   "Q13.0" := "QCC除尘管道清洗阀";
   "Q13.1" := "QCC除尘清洗阀";
   "Q13.2" := "QSS输送管路清洗阀";
   "Q13.3" := "QLC料仓清洗阀";
   "Q13.4" := "QJR加热清洗阀";
   "Q13.5" := "QWK蜗壳清洗阀";//Q6.0
   "Q13.6" := "QCF出风高效清洗阀";
   "Q13.7" := "QZT主塔排水阀";

   "Q14.0" := "QSS输送管路排水阀";
   "Q14.1" := "QLC料仓清洗排水阀";
   "Q14.2" := "QSF送风机清洗阀";
   "Q14.3" := "QYF引风机清洗阀";
   "Q14.4" := "QYJ一级冷凝清洗阀";
   "Q14.5" := "QEJ二级冷凝清洗阀";
   "Q14.6" := "QSF送风机排水阀";
   "Q14.7" := "QYF引风机排水阀";

   "Q15.0" :="QYJ一级旋风振打锤" ;//主塔振打1
   "Q15.1" :="QYJ一级旋风振荡器" ;//主塔振打2
   "Q15.2" := "QEJ二级旋风振打锤";//主塔振打3
   "Q15.3" :="QZT主塔气锤4" ;//主塔振打4
   "Q15.4" :="QQZ前置水阀" ;//布袋振打1
   //"Q15.5" :="QSB设备振打" ;//布袋振打2
   (* "Q15.6" :="QBD布袋振打3" ;//布袋振打3
   "Q15.7" :="QBD布袋振打4" ;//布袋振打4 *)

   "Q15.6" :="QYH氧含仪隔断阀" ;//氧含仪隔断阀1
   "Q15.7" :="QHS回水隔断阀1" ;//这个空的



   //QW

   "QW100" := "QWFK放空比例调节阀";
   "QW102" := "QWJF进风加热比例调节阀";
   "QW104" := "QWHF回风加热比例调节阀";

   "QW108" := "QWSF送风机";
   "QW110" := "QWYF引风机";
   "QW112" := "QWLX离心雾化器";
   "QW114" := "QWJL进料泵";


   //IW 

   "IWJF进风流量计" := "IW100";
   "IWJL进料流量" := "IW102";
   "IWJF进风压差变送器" := "IW104";
   "IWCF出风高效压差变送器" := "IW106";

   "IWBD布袋压差变送器" := "IW108";
   "IWSS输送高效压差变送器" := "IW110";
   "IWJL进料压力" := "IW112";
   "IWTN塔内压力" := "IW114";

   "IWGD管道压力变送器" := "IW116";
   "IWJD进氮压力" := "IW118";
   "IWFK放空比例反馈" := "IW120";
   "IWJF进风加热比例反馈" := "IW122";

   "IWHF回风加热比例反馈" := "IW124";
   "IWWH雾化油压" := "IW126";
   "IWYH氧含仪1" := "IW128";
   "IWYH氧含仪2" := "IW130";

   //第二个模块
   "IWYJ一级溶剂液位计" := "IW132";
   "IWEJ二级溶剂液位计" := "IW134";
   "IWCW除雾溶剂液位计" := "IW136";
   "IWFD阀岛气压" := "IW138";

   "IWQZ前置水罐液位计" := "IW140";
   "IWBY备用2" := "IW142";
   "IWBY备用3" := "IW144";
   "IWBY备用4" := "IW146";


   //IW140-IW146空。
   "IWBY备用5" := "IW148";
   "IWSF送风机" := "IW150";
   "IWYF引风机" := "IW152";
   "IWLX离心雾化器" := "IW154";

   "IWJL进料泵" := "IW156";
   "IWBY备用6" := "IW158";
   "IWBY备用7" := "IW160";
   "IWBY备用8" := "IW162";
END_REGION
END_FUNCTION

FUNCTION_BLOCK "A8-通信心跳"   // FB31, SCL
{ S7_Optimized_Access := 'TRUE' }
VERSION : 0.1
// stored: AutoNumber true, IsIECCheckEnabled false, IsRetainMemResEnabled false, MemoryReserve 100, SetENOAutomatically false, UDAEnableTagReadback false
   VAR_INPUT
      XH信号超时报警 : Real := 120.0;   // SB设备写读与创造写对比,如果不同超时,即判断报警
   END_VAR
   VAR_OUTPUT
      设备未通信报警 : Bool;
   END_VAR
   VAR_IN_OUT
      SB设备写读 : Real;
      SB设备写 : Real;
      SB设备写检测 : Real;
   END_VAR
   VAR RETAIN
      MC脉冲切换时间 : Real := 20.0;   // 给写信号+1,创造不同，10秒切换一次
   END_VAR
   VAR
      XH信号不同超时报警 : Real := 120.0;   // SB设备写读与创造写对比,如果不同超时,即判断报警
      XH信号相同超时报警 : Real := 120.0;   // SB设备写读与创造写对比,如果相同超时,即判断报警
      TON1 { S7_SetPoint := 'True'} : TON_TIME;
      TON1ET { S7_SetPoint := 'True'} : Time;
      TON2 : TON_TIME;
      TON2ET { S7_SetPoint := 'True'} : Time;
      LS设备通延辅助1 { S7_SetPoint := 'True'} : Bool;
      LS设备通延辅助2 : Bool;
      LS通信脉冲读1 : Bool;
      LS通信脉冲读2 : Bool;
      LS设备读温比较 : Real;
      T1S : TON_TIME;
      YC1 { S7_SetPoint := 'True'} : Real;
   END_VAR
   VAR_TEMP
      "m" : Int;
   END_VAR
BEGIN
   IF "FirstScan" THEN
       RESET_TIMER(#TON1);
       RESET_TIMER(#TON2);
       #LS设备通延辅助1 := 0;
       #LS设备通延辅助2 := 0;
   END_IF;

   #XH信号不同超时报警:=#XH信号超时报警;
   #XH信号相同超时报警 := #XH信号超时报警;
   #MC脉冲切换时间 := 20;

   IF #T1S.Q AND #YC1<#MC脉冲切换时间 THEN
       #YC1 := #YC1 + 1;
   END_IF;

   IF #YC1 >= #MC脉冲切换时间 THEN
       #YC1 := 0;
   END_IF;

   IF #YC1 <= (#MC脉冲切换时间 - 10) THEN

       #LS通信脉冲读1 := 1;
       #LS通信脉冲读2 := 0;
   ELSE
       #LS通信脉冲读1 := 0;
       #LS通信脉冲读2 := 1;
   END_IF;

   IF #LS通信脉冲读1 THEN
       //冷水
       #LS设备读温比较 := #SB设备写读;
       #SB设备写检测 := #SB设备写 + 0.1;
       #TON1(IN := (ABS(#LS设备读温比较) <> ABS(#SB设备写检测)),
             PT := DINT_TO_TIME(REAL_TO_DINT(#XH信号不同超时报警 * 1000.0)),
             Q => #LS设备通延辅助1,
             ET => #TON1ET);

      #TON2(IN := (ABS(#LS设备读温比较) = ABS(#SB设备写检测)),
             PT := DINT_TO_TIME(REAL_TO_DINT(#XH信号相同超时报警 * 1000.0)),
             Q => #LS设备通延辅助2,
             ET => #TON2ET);

   END_IF;

   IF #LS通信脉冲读2 AND NOT #LS通信脉冲读1 THEN
       #SB设备写检测 := #SB设备写;
   END_IF;

   IF #LS设备通延辅助1 OR #LS设备通延辅助2  THEN
       #设备未通信报警 := 1;
   ELSE
       #设备未通信报警 := 0;
   END_IF;

   #T1S(IN := NOT #T1S.Q,
       PT := T#1S);
END_FUNCTION_BLOCK

FUNCTION_BLOCK "0-模拟量滤波"   // FB109, LAD
{ S7_Optimized_Access := 'TRUE' }
VERSION : 0.1
// stored: AutoNumber true, IsIECCheckEnabled false, IsRetainMemResEnabled false, MemoryReserve 100, SetENOAutomatically false, UDAEnableTagReadback false
   VAR_INPUT
      模拟量数据输入 : Int;
      "上限(工程量)" : Real;
      "下限(工程量)" : Real := 100.0;
      "采样时间间隔（秒）" : Real := 1.0;
      滤波强度 : Int := 10;
   END_VAR
   VAR_OUTPUT
      工程量数据输出 : Real;
      "工程量数据输出(滤波后)" : Real;
      Error_MAX : Bool;
      Error_MIN : Bool;
   END_VAR
   VAR
      AI : Int;
      "Time" : Time;
      T0 { S7_SetPoint := 'True'} : TON_TIME;
      T1 { S7_SetPoint := 'True'} : TON_TIME;
      P0 { S7_SetPoint := 'True'} : R_TRIG;
      LB { S7_SetPoint := 'True'} : Array[1..20] of Real;
      ZS : Real;
      N : Int;
      stat滤波强度 : Int;
   END_VAR
BEGIN

REGION Network 1 (SCL)
   #Time:=DINT_TO_TIME( REAL_TO_DINT( #"采样时间间隔（秒）"*1000.0)-10);
   #T0(IN:=NOT #T1.Q,
       PT:=#Time);
   #T1(IN:=#T0.Q,
       PT:=T#10MS);
   #P0(CLK:=#T0.Q);



   #AI := #模拟量数据输入;
   IF #AI<0 THEN
       #AI := 0;
       #Error_MIN := 1;
   ELSE
       #Error_MIN := 0;
       ;
   END_IF;

   IF #AI>27648 THEN
       #AI := 27648;
       #Error_MAX := 1;
   ELSE
       #Error_MAX := 0;
       ;
   END_IF;
   #stat滤波强度 := #滤波强度;
   IF #滤波强度 > 20 THEN
       #stat滤波强度 := 20;
   END_IF;
   IF #滤波强度 < 1 THEN
       #stat滤波强度 := 1;
   END_IF;

   IF #P0.Q THEN
       #工程量数据输出 := INT_TO_REAL(#AI) / 27648.0 * (#"上限(工程量)" - #"下限(工程量)") + #"下限(工程量)";
       FOR #N := #stat滤波强度 TO 2 BY -1 DO
           #LB[#N] := #LB[#N - 1];
           ;
       END_FOR;
       #LB[1] := #工程量数据输出;

       #ZS := 0;
       FOR #N := 1 TO #stat滤波强度 DO
           #ZS := #ZS + #LB[#N];
       END_FOR;


       #"工程量数据输出(滤波后)" := #ZS / #stat滤波强度;



   END_IF;
END_REGION
END_FUNCTION_BLOCK

FUNCTION_BLOCK "0-模拟量滤波简"   // FB86, SCL
{ S7_Optimized_Access := 'TRUE' }
VERSION : 0.1
// stored: AutoNumber true, IsIECCheckEnabled false, IsRetainMemResEnabled false, MemoryReserve 100, SetENOAutomatically false, UDAEnableTagReadback false
   VAR_INPUT
      输入 : Real;   // 转换后的模拟量输入端
      采集时间 : Time := T#200ms;   // 多长时间采集一次数据，单位ms
      模式 : Bool;   // false为算数平均滤波，true为切头尾平均滤波
   END_VAR
   VAR_OUTPUT
      输出 : Real;   // 滤波后的输出值
   END_VAR
   VAR_IN_OUT
      滤波强度 : Int := 3;   // 多少个数据平均一次
   END_VAR
   VAR
      T0 : TON_TIME;
      T1 { S7_SetPoint := 'True'} : TON_TIME;
      P { S7_SetPoint := 'True'} : R_TRIG;
      最小值 { S7_SetPoint := 'True'} : Real;
      最大值 : Real;
      中间寄存数值 : Array[0..30] of Real;
   END_VAR
   VAR_TEMP
      "a" : DInt;
      "b" : DInt;
      总和 : Real;
   END_VAR
BEGIN
   REGION 初始化
       #最大值 := #中间寄存数值[1];
       #最小值 := #中间寄存数值[1];
   END_REGION


   REGION 滤波强度限制
       IF #滤波强度 < 3 THEN
           #滤波强度 := 3;
       END_IF;
       IF #滤波强度 > 30 THEN
           #滤波强度 := 30;
       END_IF;
   END_REGION


   REGION 构速时钟脉冲
       #T0(IN := NOT #T1.Q,
           PT := #采集时间 - T#20MS);
       #T1(IN :=  #T0.Q,
           PT := T#20MS);
       #P(CLK := #T0.Q);
   END_REGION

   REGION 数据写入
       IF #P.Q THEN
           FOR #a := #滤波强度 TO 2 BY -1 DO //依次将输入数据存入到寄存数组中
               #中间寄存数值[#a] := #中间寄存数值[#a - 1];
           END_FOR;
           #中间寄存数值[1] := #输入;
       END_IF;
   END_REGION


   REGION 找最值以及计算总和
       FOR #b := 1 TO #滤波强度 DO
           IF #中间寄存数值[#b] > #最大值 THEN
               #最大值 := #中间寄存数值[#b];
           END_IF;
           IF #中间寄存数值[#b] < #最小值 THEN
               #最小值 := #中间寄存数值[#b];
           END_IF;
           #总和 := #总和 + #中间寄存数值[#b]; //计算总和
       END_FOR;
   END_REGION


   REGION 求平均以及输出
       IF #模式 = TRUE THEN
           #输出 := (#总和 - #最大值 - #最小值) / DINT_TO_REAL((#滤波强度) - 2);//切尾平均滤波后输出
       ELSE
           #输出 := #总和 / DINT_TO_REAL(#滤波强度);//算数平均输出
       END_IF;
   END_REGION
END_FUNCTION_BLOCK

FUNCTION_BLOCK "0-模拟量输入"   // FB35, SCL
{ S7_Optimized_Access := 'TRUE' }
VERSION : 0.1
// stored: AutoNumber true, IsIECCheckEnabled false, IsRetainMemResEnabled false, MemoryReserve 100, SetENOAutomatically false, UDAEnableTagReadback false
   VAR_INPUT
      模拟量数据输入 : Int;
      上限模拟 : Real := 27648.0;
      下限模拟 : Real := 5530.0;
      上限工程 : Real := 100.0;
      下限工程 : Real := 0.0;
      修正值 : Real;
      错误确认 : Bool;
      高高限工程量 : Real := 90.0;
      高限工程量 : Real := 80.0;
      低限工程量 : Real := 20.0;
      低低限工程量 : Real := 10.0;
      高高限位滤波时间设定 : Time := T#1s;
      高限位滤波时间设定 : Time := T#1s;
      低限位滤波时间设定 : Time := T#1s;
      低低限位滤波时间设定 : Time := T#1s;
      MODE : Byte := 16#1;   // 0报警输出不自动消除，1报警情况结束自动消除 2.高高或低低限位保持报警，其余自动确认报警
   END_VAR
   VAR_OUTPUT
      工程量数据输出 : Real;
      断线错误 : Bool;
      超过高高限位 : Bool;
      超过高限位 : Bool;
      低于低限位 : Bool;
      低于低低限位 : Bool;
   END_VAR
   VAR
      临时模拟量数据输入 : Real;
      缩放比例 : Real;
      T : Struct
         高高限位滤波时间 { S7_SetPoint := 'True'} : TON_TIME;
         高限位滤波时间 { S7_SetPoint := 'True'} : TON_TIME;
         低限位滤波时间 { S7_SetPoint := 'True'} : TON_TIME;
         低低限位滤波时间 { S7_SetPoint := 'True'} : TON_TIME;
      END_STRUCT;
   END_VAR
BEGIN
   #临时模拟量数据输入 := INT_TO_REAL(#模拟量数据输入);  //将模拟量输入转换为real类型
   // IF #临时模拟量数据输入 > #模拟量Max THEN
   //     #临时模拟量数据输入 := #模拟量Max;
   // END_IF;
   // IF #临时模拟量数据输入 < #模拟量Min THEN
   //     #临时模拟量数据输入 := #模拟量Min;
   // END_IF;
   #缩放比例 := (#上限工程 - #下限工程) / (#上限模拟 - #下限模拟);//算出实际值与模拟量的缩放比例
   #工程量数据输出 := (#模拟量数据输入 - #下限模拟) * #缩放比例 + #下限工程+#修正值;      //转换完成


   //2
   //
   IF (#临时模拟量数据输入 > 30000 OR #临时模拟量数据输入 < 4000 )
       AND NOT #错误确认 THEN
       #断线错误 := 1;
   ELSE
       #断线错误 := 0;
   END_IF;

   //3
   //

   #T.高高限位滤波时间(IN := #工程量数据输出 > #高高限工程量,
               PT := #高高限位滤波时间设定);
   IF #T.高高限位滤波时间.Q OR (#超过高高限位 AND (#MODE = 0 OR #MODE = 2)) AND NOT #错误确认 THEN

       #超过高高限位 := 1;
   ELSE
       #超过高高限位 := 0;
   END_IF;

   (* IF #超过高高限位 AND (#MODE = 0 OR #MODE = 2) AND NOT #错误确认 THEN
       #超过高高限位 := 1;
   ELSE
       #超过高高限位 := 0;
   END_IF; *)

   //4
   //
   #T.高限位滤波时间(IN := #工程量数据输出 >= #高限工程量,
              PT := #高限位滤波时间设定);
   IF #T.高限位滤波时间.Q OR (#超过高限位 AND #MODE = 0) AND NOT #错误确认 THEN
       #超过高限位 := 1;
   ELSE
       #超过高限位 := 0;
   END_IF;

   //5
   //
   #T.低限位滤波时间(IN := #工程量数据输出 <= #低限工程量,
              PT := #低限位滤波时间设定);

   IF #T.低限位滤波时间.Q OR (#低于低限位 AND #MODE = 0) AND NOT #错误确认 THEN
       #低于低限位 := 1;
   ELSE
       #低于低限位 := 0;
   END_IF;

   (* IF #低于低限位 AND #MODE=0 THEN
       #低于低限位 := 1;
   ELSE
       #低于低限位 := 0;
   END_IF; *)

   //6
   //
   #T.低低限位滤波时间(IN := #工程量数据输出 <= #低低限工程量,
               PT := #低低限位滤波时间设定);
   IF #T.低低限位滤波时间.Q OR (#低于低低限位 AND (#MODE = 0 OR #MODE = 2)) AND NOT #错误确认 THEN
       #低于低低限位 := 1;
   ELSE
       #低于低低限位 := 0;
   END_IF;

   (* IF #低于低低限位 AND (#MODE=0 OR #MODE=2) AND NOT #错误确认  THEN
       #低于低低限位 := 1;
   ELSE
       #低于低低限位 := 0;
   END_IF; *)
END_FUNCTION_BLOCK

FUNCTION_BLOCK "0-模拟量输入1PID"   // FB172, LAD
{ S7_Optimized_Access := 'TRUE' }
VERSION : 0.1
// stored: AutoNumber true, IsIECCheckEnabled false, IsRetainMemResEnabled false, MemoryReserve 100, SetENOAutomatically false, UDAEnableTagReadback false
   VAR_INPUT
      "仪表反馈值(模拟量)" : Int;
      积分P : Real := 0.5;
      微分I : Real := 0.5;
      "上限(模拟量)" : Real := 27648.0;
      "下限(模拟量)" : Real;
      "上限(工程量)" : Real := 200.0;
      "下限(工程量)" : Real;
      "设定补偿值(工程量)" : Real := 0.5;   // PID值快到达设定值时由于PID调节作用始终差一点才能到达设定值，所以用补偿的方式直接加上
      "设定目标值(工程量)" : Real := 100.0;
   END_VAR
   VAR_OUTPUT
      "仪表反馈值(工程量)" : Real;   // 由模拟量输入直接比例缩放转出的工程量，作用就是看一下显示
      "给定变频器(模拟量)" : Int;   // PID调节后的直接给变频器的模拟量值0-27648
      "PID调节输出值(工程量)" : Real;
   END_VAR
   VAR
      临时模拟量数据输入 : Real;
      缩放比例 : Real;
      实际模拟量 : Real;
      当前偏差 : Real;
      上一次偏差 : Real;
      输出控制量 : Real;
      PQW : Real;
   END_VAR
BEGIN

REGION Network 1 (SCL)
   //模拟量转换工程值
   #临时模拟量数据输入 := INT_TO_REAL(#"仪表反馈值(模拟量)");  //将模拟量输入转换为real类型
   #缩放比例 := (#"上限(工程量)" - #"下限(工程量)") / (#"上限(模拟量)" - #"下限(模拟量)");//算出实际值与模拟量的缩放比例
   #"仪表反馈值(工程量)" := (#"仪表反馈值(模拟量)"-#"下限(模拟量)") * #缩放比例+#"下限(工程量)";      //转换完成
   #当前偏差 := #"设定目标值(工程量)" - #"仪表反馈值(工程量)";

   //PID计算
   IF  #"设定补偿值(工程量)">ABS( #当前偏差) THEN
       #输出控制量 := 0;
   ELSIF #"设定补偿值(工程量)"<ABS( #当前偏差) THEN
       #输出控制量 := #积分P*(#当前偏差-#上一次偏差)+#微分I*#当前偏差;
   END_IF;

   #"PID调节输出值(工程量)":=#输出控制量;

   //上下限制
   IF #"PID调节输出值(工程量)"> #"上限(工程量)"THEN
       #"PID调节输出值(工程量)" := #"上限(工程量)";
   ELSIF #"PID调节输出值(工程量)"< #"下限(工程量)"THEN
       #"PID调节输出值(工程量)" := #"下限(工程量)";
   END_IF;


   //控制电机输出

   #上一次偏差 := #当前偏差;
   #PQW:=(#"PID调节输出值(工程量)"-#"下限(工程量)")/(#"上限(工程量)"-#"下限(工程量)")*#"上限(模拟量)";
   #"给定变频器(模拟量)" := REAL_TO_INT(#PQW);
END_REGION
END_FUNCTION_BLOCK

FUNCTION_BLOCK "0-模拟量输入2PID"   // FB79, SCL
{ S7_Optimized_Access := 'TRUE' }
VERSION : 0.1
// stored: AutoNumber true, IsIECCheckEnabled false, IsRetainMemResEnabled false, MemoryReserve 100, SetENOAutomatically false, UDAEnableTagReadback false
   VAR_INPUT
      AM : Bool := TRUE;   // 手动调节: 0,手动; 1,自动.
      ManualValue : Real;   // 手动调节输出值:0-100%.
      Enable : Bool;   // 自动调节使能. 1,启用; 0,不启用.
      Mode : Int := 1;   // 控制模式: 0,制热;1,制冷; 2,输出0.
      Setpoint : Real;   // 控制目标值
      Input : Real;   // 控制实际值
      ControlledObject_FB : Real;   // 受控对象实际值反馈(开度/频率...)
      Kp : Real;   // 比例系数(大于零实数)
      DeadZone : Real;   // 死区
      MAX : Real := 100.0;   // 上限
      MIN : Real;   // 下限
   END_VAR
   VAR_OUTPUT
      Output : Real;   // 受控对象输出值
   END_VAR
   VAR
      AutoValue : Real;
      output_Temp { ExternalAccessible := 'False'; ExternalVisible := 'False'; ExternalWritable := 'False'} : Real;
      RT_C : DInt;
   END_VAR
BEGIN
   IF  #AM AND #Enable THEN
       IF (#Mode=1) AND (ABS(#Input - #Setpoint) > #DeadZone) THEN
           #AutoValue := #ControlledObject_FB + #Kp * (#Input - #Setpoint) / 100;
       ELSIF (#Mode=0) AND (ABS(#Input - #Setpoint) > #DeadZone) THEN
           #AutoValue := #ControlledObject_FB - #Kp * (#Input - #Setpoint) / 100;
       ELSIF (#Mode=2) THEN
           #AutoValue := 0;
       ELSE
           #AutoValue := #ControlledObject_FB;
       END_IF;
   END_IF;

   IF NOT #AM THEN
       #output_Temp := #ManualValue;
   ELSE
       #output_Temp := #AutoValue;
   END_IF;

   IF #output_Temp >= #MAX THEN
       #Output := #MAX;
   ELSIF #output_Temp <= #MIN THEN
       #Output := #MIN;
   ELSE
       #Output := #output_Temp;
   END_IF;
END_FUNCTION_BLOCK

FUNCTION_BLOCK "0-模拟量输入压差"   // FB69, SCL
{ S7_Optimized_Access := 'TRUE' }
VERSION : 0.1
// stored: AutoNumber true, IsIECCheckEnabled false, IsRetainMemResEnabled false, MemoryReserve 100, SetENOAutomatically false, UDAEnableTagReadback false
   VAR_INPUT
      模拟量数据输入 : Int;
      上限模拟 : Real := 27648.0;
      下限模拟 : Real := 5530.0;
      上限工程 : Real := 100.0;
      下限工程 : Real := 0.0;
      修正值 : Real;
      错误确认 : Bool;
      高高限工程量 : Real := 90.0;
      高限工程量 : Real := 80.0;
      低限工程量 : Real := 20.0;
      低低限工程量 : Real := 10.0;
      高高限位滤波时间设定 : Time := T#1s;
      高限位滤波时间设定 : Time := T#1s;
      低限位滤波时间设定 : Time := T#1s;
      低低限位滤波时间设定 : Time := T#1s;
      MODE : Byte := 16#1;   // 0报警输出不自动消除，1报警情况结束自动消除 2.高高或低低限位保持报警，其余自动确认报警
   END_VAR
   VAR_OUTPUT
      工程量数据输出 : Real;
      断线错误 : Bool;
      超过高高限位 : Bool;
      超过高限位 : Bool;
      低于低限位 : Bool;
      低于低低限位 : Bool;
   END_VAR
   VAR_IN_OUT
      风机 : Bool;
   END_VAR
   VAR
      临时模拟量数据输入 : Real;
      缩放比例 : Real;
      T : Struct
         高高限位滤波时间 { S7_SetPoint := 'True'} : TON_TIME;
         高限位滤波时间 { S7_SetPoint := 'True'} : TON_TIME;
         低限位滤波时间 { S7_SetPoint := 'True'} : TON_TIME;
         低低限位滤波时间 { S7_SetPoint := 'True'} : TON_TIME;
      END_STRUCT;
   END_VAR
BEGIN
   #临时模拟量数据输入 := INT_TO_REAL(#模拟量数据输入);  //将模拟量输入转换为real类型
   // IF #临时模拟量数据输入 > #模拟量Max THEN
   //     #临时模拟量数据输入 := #模拟量Max;
   // END_IF;
   // IF #临时模拟量数据输入 < #模拟量Min THEN
   //     #临时模拟量数据输入 := #模拟量Min;
   // END_IF;
   #缩放比例 := (#上限工程 - #下限工程) / (#上限模拟 - #下限模拟);//算出实际值与模拟量的缩放比例
   #工程量数据输出 := (#模拟量数据输入 - #下限模拟) * #缩放比例 + #下限工程+#修正值;      //转换完成


   //2
   //
   IF (#临时模拟量数据输入 > 30000 OR #临时模拟量数据输入 < 4000 OR #断线错误)
       AND NOT #错误确认 THEN
       #断线错误 := 1;
   ELSE
       #断线错误 := 0;
   END_IF;

   //3
   //

   #T.高高限位滤波时间(IN := #工程量数据输出 > #高高限工程量,
               PT := #高高限位滤波时间设定);
   IF #T.高高限位滤波时间.Q OR (#超过高高限位 AND (#MODE = 0 OR #MODE = 2)) AND NOT #错误确认 THEN

       #超过高高限位 := 1;
   ELSE
       #超过高高限位 := 0;
   END_IF;

   (* IF #超过高高限位 AND (#MODE = 0 OR #MODE = 2) AND NOT #错误确认 THEN
       #超过高高限位 := 1;
   ELSE
       #超过高高限位 := 0;
   END_IF; *)

   //4
   //
   #T.高限位滤波时间(IN := #工程量数据输出 >= #高限工程量,
              PT := #高限位滤波时间设定);
   IF #T.高限位滤波时间.Q OR (#超过高限位 AND #MODE = 0) AND NOT #错误确认 THEN
       #超过高限位 := 1;
   ELSE
       #超过高限位 := 0;
   END_IF;

   //5
   //
   #T.低限位滤波时间(IN := #工程量数据输出 <= #低限工程量,
              PT := #低限位滤波时间设定);

   IF #T.低限位滤波时间.Q OR (#低于低限位 AND #MODE = 0) AND #风机 AND NOT #错误确认 THEN
       #低于低限位 := 1;
   ELSE
       #低于低限位 := 0;
   END_IF;

   (* IF #低于低限位 AND #MODE=0 THEN
       #低于低限位 := 1;
   ELSE
       #低于低限位 := 0;
   END_IF; *)

   //6
   //
   #T.低低限位滤波时间(IN := #工程量数据输出 <= #低低限工程量,
               PT := #低低限位滤波时间设定);
   IF #T.低低限位滤波时间.Q OR (#低于低低限位 AND (#MODE = 0 OR #MODE = 2)) AND NOT #错误确认 THEN
       #低于低低限位 := 1;
   ELSE
       #低于低低限位 := 0;
   END_IF;

   (* IF #低于低低限位 AND (#MODE=0 OR #MODE=2) AND NOT #错误确认  THEN
       #低于低低限位 := 1;
   ELSE
       #低于低低限位 := 0;
   END_IF; *)
END_FUNCTION_BLOCK

FUNCTION_BLOCK "1-模拟量输出1"   // FB75, SCL
{ S7_Optimized_Access := 'TRUE' }
VERSION : 0.1
// stored: AutoNumber true, IsIECCheckEnabled false, IsRetainMemResEnabled false, MemoryReserve 100, SetENOAutomatically false, UDAEnableTagReadback false
   VAR_INPUT
      HMI上限 : Real;
      HMI下限 : Real;
      PLC上限 : Int;
      PLC下限 : Int;
   END_VAR
   VAR_IN_OUT
      PLC调控 : Int;
      HMI设定 : Real;
   END_VAR
   VAR
      DBD1 : Real;
   END_VAR
BEGIN
   #DBD1 := NORM_X_REAL(MIN := #HMI下限, VALUE := #HMI设定, MAX := #HMI上限);
   #PLC调控 := SCALE_X_INT(MIN := #PLC下限, VALUE := #DBD1, MAX := #PLC上限);
END_FUNCTION_BLOCK

FUNCTION_BLOCK "1-模拟量输出2"   // FB77, SCL
{ S7_Optimized_Access := 'TRUE' }
VERSION : 0.1
// stored: AutoNumber true, IsIECCheckEnabled false, IsRetainMemResEnabled false, MemoryReserve 100, SetENOAutomatically false, UDAEnableTagReadback false
   VAR_INPUT
      R_Max : Real;
      R_Min : Real;
      R_Value : Real;
   END_VAR
   VAR_OUTPUT
      I_ChValue : Int;
   END_VAR
BEGIN
   (**)
   #I_ChValue := REAL_TO_INT((#R_Value - #R_Min) / (#R_Max - #R_Min) * 27648.0);
END_FUNCTION_BLOCK

FUNCTION_BLOCK "3-延时开关M"   // FB78, SCL
{ S7_Optimized_Access := 'TRUE' }
VERSION : 0.1
// stored: AutoNumber true, IsIECCheckEnabled false, IsRetainMemResEnabled false, MemoryReserve 100, SetENOAutomatically false, UDAEnableTagReadback false
   VAR_INPUT
      B_IN : Bool;   // 启动/关闭信号输入
      T_IN : Int;   // 延时时间(单位:分)
      B_Status : Bool;   // 运行状态
   END_VAR
   VAR_OUTPUT
      B_OUT : Bool;   // 启动/关闭信号输出
   END_VAR
   VAR
      RT1 { S7_SetPoint := 'True'} : R_TRIG;   // 计时_1S
      i : UDInt;
   END_VAR
BEGIN
   (*水泵关机延时功能:
       1.立即开机
       2.延时I_IN分钟后关闭
       3.延时关机期间如果水泵手动/其他原因关闭,延时时间清零,立即关闭
   *)

   #RT1(CLK:="Clock_1Hz");

   IF NOT #B_IN THEN
       IF #RT1.Q THEN
           #i += 1;
       END_IF;
   ELSE
       #i := 0;
   END_IF;

   IF #B_IN THEN
       #B_OUT := 1;    //立即开
   ELSIF NOT #B_IN AND #i >= #T_IN * 60 THEN    //延时关
       #B_OUT := 0;
   ELSIF NOT #B_IN AND #i < #T_IN * 60 AND  #B_Status THEN  //延时关机期间如果水泵手动/其他原因关闭,延时时间清零,立即关闭
       #B_OUT := 0;
   END_IF;
END_FUNCTION_BLOCK

FUNCTION_BLOCK "3-延时开关S"   // FB73, SCL
{ S7_Optimized_Access := 'TRUE' }
VERSION : 0.1
// stored: AutoNumber true, IsIECCheckEnabled false, IsRetainMemResEnabled false, MemoryReserve 100, SetENOAutomatically false, UDAEnableTagReadback false
   VAR_INPUT
      B_IN : Bool;   // 启动/关闭信号输入
      T_IN : Int;   // 延时时间(单位:秒)
      B_Status : Bool;   // 运行状态
   END_VAR
   VAR_OUTPUT
      B_OUT : Bool;   // 启动/关闭信号输出
   END_VAR
   VAR
      R_TRIG_1 { S7_SetPoint := 'True'} : R_TRIG;   // 计时_1S
      i : UDInt;
   END_VAR
BEGIN
   (*水泵关机延时功能:
       1.立即开机
       2.延时I_IN分钟后关闭
       3.延时关机期间如果水泵手动/其他原因关闭,延时时间清零,立即关闭
   *)

   #R_TRIG_1(CLK:="Clock_1Hz");

   IF NOT #B_IN THEN
       IF #R_TRIG_1.Q THEN
           #i += 1;
       END_IF;
   ELSE
       #i := 0;
   END_IF;

   IF #B_IN THEN
       #B_OUT := 1;    //立即开
   ELSIF NOT #B_IN AND #i >= #T_IN  THEN    //延时关
       #B_OUT := 0;
   ELSIF NOT #B_IN AND #i < #T_IN  AND  #B_Status THEN  //延时关机期间如果水泵手动/其他原因关闭,延时时间清零,立即关闭
       #B_OUT := 0;
   END_IF;
END_FUNCTION_BLOCK

FUNCTION_BLOCK "4-点斜率输入->输出"   // FB64, LAD
{ S7_Optimized_Access := 'TRUE' }
VERSION : 0.1
// stored: AutoNumber true, IsIECCheckEnabled false, IsRetainMemResEnabled false, MemoryReserve 100, SetENOAutomatically false, UDAEnableTagReadback false
   VAR_INPUT
      sr输入ok : Real;
   END_VAR
   VAR_OUTPUT
      sc输出ok : Int;
   END_VAR
   VAR_IN_OUT
      sr输入1 : Real;
      sc输出1 : Real;
      sr输入2 : Real;
      sc输出2 : Real;
   END_VAR
BEGIN

REGION Network 1 (SCL)


   #sc输出ok := REAL_TO_INT(((#sc输出2 - #sc输出1) / (#sr输入2 - #sr输入1)) * #sr输入ok);
END_REGION
END_FUNCTION_BLOCK

FUNCTION_BLOCK "4-点斜率输出->输入"   // FB68, LAD
{ S7_Optimized_Access := 'TRUE' }
VERSION : 0.1
// stored: AutoNumber true, IsIECCheckEnabled false, IsRetainMemResEnabled false, MemoryReserve 100, SetENOAutomatically false, UDAEnableTagReadback false
   VAR_INPUT
      sc输出ok : Int;
   END_VAR
   VAR_OUTPUT
      sr输入ok : Real;
   END_VAR
   VAR_IN_OUT
      sr输入1 : Real;
      sc输出1 : Real;
      sr输入2 : Real;
      sc输出2 : Real;
   END_VAR
BEGIN

REGION Network 1 (SCL)


   #sr输入ok := REAL_TO_INT(((#sr输入2 - #sr输入1)/(#sc输出2 - #sc输出1) ) * #sc输出ok);
END_REGION
END_FUNCTION_BLOCK

FUNCTION_BLOCK "5-定时器"   // FB72, SCL
{ S7_Optimized_Access := 'TRUE' }
VERSION : 0.1
// stored: AutoNumber true, IsIECCheckEnabled false, IsRetainMemResEnabled false, MemoryReserve 100, SetENOAutomatically false, UDAEnableTagReadback false
   VAR_INPUT
      计时开始 : Bool;
      定时器设置时间 : Time;
   END_VAR
   VAR_OUTPUT
      剩余时间分 : Int;
      剩余时间秒 : Int;
      计时到达 : Bool;
   END_VAR
   VAR
      定时器当前时间 : Time;
      "TIMER" : TON_TIME;
   END_VAR
   VAR_TEMP
      TEMP剩余时间 : Time;
   END_VAR
BEGIN
   #TIMER(IN:=#计时开始,
          PT:=#定时器设置时间,
          Q=>#计时到达,
          ET=>#定时器当前时间);



   //计时未开始，剩余时间为0
   IF NOT #计时开始 THEN
       #剩余时间分 := 0;
       #剩余时间秒 := 0;
   END_IF;

   IF #定时器当前时间 > t#0ms THEN
       #TEMP剩余时间 := (#定时器设置时间 / 1000)-(#定时器当前时间/1000);
       #剩余时间分 := TIME_TO_INT(#TEMP剩余时间)/60;
       #剩余时间秒 := TIME_TO_INT(#TEMP剩余时间) MOD 60;
   END_IF;
END_FUNCTION_BLOCK

FUNCTION_BLOCK "5-斜坡函数发生器"   // FB91, SCL
{ S7_Optimized_Access := 'TRUE' }
VERSION : 0.1
// stored: AutoNumber true, IsIECCheckEnabled false, IsRetainMemResEnabled false, MemoryReserve 100, SetENOAutomatically false, UDAEnableTagReadback false
   VAR_INPUT
      输入 : Real;
      斜坡激活 : Bool;   // 0：直接输出 1：斜坡输出
      上升斜率 : Real := 1.0;   // 斜坡上升增量值 （单位值/秒）
      下降斜率 : Real := 1.0;   // 斜坡下降增量值 （ 单位值/秒）
      输出上限 : Real := 100.0;
      输出下限 : Real := 0.0;
   END_VAR
   VAR_OUTPUT
      输出 : Real;
   END_VAR
BEGIN

   //可用于电机的速度给定以实现平滑升/降速；重要的调节阀门设定，进行平滑过度，防止水锤及工艺扰动等现象
   //在循环中断OB30中调用该FB块，OB30循环时间设置为100ms。
   //如果上升斜率设置为1/s，输入则上升斜坡将持续10s（设定值从0增加至10）。
   //公式：Y=Y+A。

   IF NOT #斜坡激活 THEN
       //直接输出
       #输出 := #输入;
   ELSE
       //斜坡输出
       IF #输入 > #输出 THEN
           //斜坡上升
           #输出 := #输出 + #上升斜率 / 10.0;
       END_IF;
       IF #输入 < #输出 THEN
           //斜坡下降
           #输出 := #输出 - #下降斜率 / 10.0;
       END_IF;
   END_IF;


   //输出限幅
   IF #输出 > #输出上限 THEN
       #输出 := #输出上限;
   END_IF;
   IF #输出 < #输出下限 THEN
       #输出 := #输出下限;
   END_IF;
END_FUNCTION_BLOCK

FUNCTION_BLOCK "5-称重法堵塞"   // FB76, LAD
{ S7_Optimized_Access := 'TRUE' }
VERSION : 0.1
// stored: AutoNumber true, IsIECCheckEnabled false, IsRetainMemResEnabled false, MemoryReserve 100, SetENOAutomatically false, UDAEnableTagReadback false
   VAR_OUTPUT
      进料堵塞辅助 : Bool;
   END_VAR
   VAR_IN_OUT
      进料蠕动泵开关 : Bool;
      当前重量值 : Real;
      上一次重量值 : Real;
      重量差值 : Real;
      称重仪实际重量 : Real;
      设定物料检测重量 : Real;
   END_VAR
BEGIN

REGION Network 1 (SCL): 初扫描 / 油炉和风机
   // 需放入Cyclic interrupt中，并设置间隔时间60000ms
   #当前重量值 := #称重仪实际重量;
   #重量差值 := #当前重量值 - #上一次重量值;
   #上一次重量值 := #称重仪实际重量;

   IF #进料蠕动泵开关 AND #重量差值 <= #设定物料检测重量 THEN
       #进料堵塞辅助 := true;
   END_IF;
END_REGION
END_FUNCTION_BLOCK

FUNCTION_BLOCK "6-系统时间读取与设置"   // FB3009, LAD
{ S7_Optimized_Access := 'FALSE' }
VERSION : 0.1
// stored: AutoNumber true, IsIECCheckEnabled false, SetENOAutomatically false, UDAEnableTagReadback false
   VAR_INPUT
      系统时间设置 : Bool;   // 时间设置按钮
      要写入的系统时间 : Date_And_Time := DT#2022-07-27-00:00:00;   // 设定时间
   END_VAR
   VAR_OUTPUT
      系统时间 : Date_And_Time;   // 系统时间
      Year : Byte;   // 年
      Month : Byte;   // 月
      Day : Byte;   // 日
      Hour : Byte;   // 时
      Minute : Byte;   // 分
      Second : Byte;   // 秒
   END_VAR
   VAR DB_SPECIFIC
      SetTimeTP1 : Byte;
      SetTimeTP2 : Byte;
      SetTimeTP3 : Byte;
      SetTimeTP4 : Byte;
      SetTimeTP5 : Byte;
      SetTimeTP6 : Byte;
      SetTimeTP7 : Byte;
      SetTimeTP8 : Byte;
      SetTimeTP9 : Date;
      SetTimeTP10 : Time_Of_Day;
   END_VAR
   VAR_TEMP
      Ret : Int;
   END_VAR
BEGIN

REGION Network 1: 读出系统时间
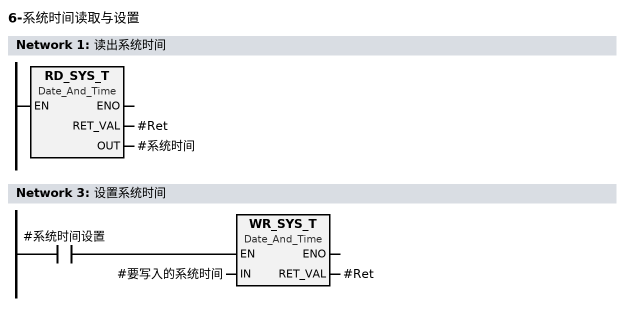
   RUNG wire#powerrail
      { S7_Templates := "date_type := Date_And_Time" } RD_SYS_T(RET_VAL => #Ret, OUT => #系统时间)
   END_RUNG
   // the same network as SCL:
   #Ret := RD_SYS_T(OUT => #系统时间);
END_REGION

NETWORK
TITLE = 读取时间

      L     %DIB10;
      T     #Year;
      L     %DIB11;
      T     #Month;
      L     %DIB12;
      T     #Day;
      L     %DIB13;
      T     #Hour;
      L     %DIB14;
      T     #Minute;
      L     %DIB15;
      T     #Second;


REGION Network 3: 设置系统时间
   RUNG wire#powerrail
      Contact( #系统时间设置 )
      { S7_Templates := "date_type := Date_And_Time" } WR_SYS_T(IN := #要写入的系统时间, RET_VAL => #Ret)
   END_RUNG
   // the same network as SCL:
   IF #系统时间设置 THEN #Ret := WR_SYS_T(IN := #要写入的系统时间); END_IF;
END_REGION
END_FUNCTION_BLOCK

FUNCTION_BLOCK "7-PID仿真LSim_PT3"   // FB80, SCL
{ S7_Optimized_Access := 'TRUE' }
VERSION : 2.1
// stored: AutoNumber true, IsIECCheckEnabled false, IsRetainMemResEnabled false, MemoryReserve 100, SetENOAutomatically false, UDAEnableTagReadback false
   VAR_INPUT
      input : Real;   // input variable
      tmLag1 : Real := 29.0;   // time lag 1 in s
      tmLag2 : Real := 17.5;   // time lag 2 in s
      tmLag3 : Real := 3.1;   // time lag 3 in s
      gain : Real := 1.0;   // proportional gain
      disturb : Real;   // disturbance variable (additional to "input")
      cycle : Real := 0.1;   // sample time [in sec]
      reset : Bool;   // complete restart (#output = #input)
   END_VAR
   VAR_OUTPUT
      error : Bool;   // error (#tmLag1 <= 0 or #tmLag2 <= 0 or #tmLag3 <= 0)
      status : Word;   // status (if #error = TRUE then status = 16#8001)
      output : Real;   // output signal (if #error = FALSE)
   END_VAR
   VAR
      statFback1 : Real;   // feedback path value 1
      statFback2 : Real;   // feedback path value 2
      statFback3 : Real;   // feedback path value 3
   END_VAR
   VAR_TEMP
      tempHvar : Real;   // help variable
      tempCycleR : Real;   // cycle to real
      tempTmLag1R : Real;   // time lag 1 to real
      tempTmLag2R : Real;   // time lag 2 to real
      tempTmLag3R : Real;   // time lag 3 to real
      tempOutvNew : Real;   // new output variable
   END_VAR
BEGIN
   //=============================================================================
   //SIEMENS AG
   //(c)Copyright 2017 All Rights Reserved
   //-----------------------------------------------------------------------------
   //Library:       Library for Controlled System Simulation
   //Tested with:   S7-1500 FW V2.0 / S7-1200 FW V4.2
   //Engineering:   STEP 7 V14 Upd2 (TIA Portal)
   //Restrictions:  Cyclic interrupt
   //Requirements:  memory card needed for S7-1500
   //Functionality: Simulation of an PT3-system
   //
   //                               gain
   //  F(p) = ------------------------------------------------------
   //         (tmLag1 * p + 1) * (tmLag2 * p + 1) * (tmLag3 * p + 1)
   //          
   //  Call the simulation in a cyclic interrupt with
   //  cyclic interrupt time at least = tmLag1/10!
   //-----------------------------------------------------------------------------
   //Change log table:
   //Version  Date       Expert in charge                Changes applied
   //02.00.00 03.02.2016 Siemens Industry Online Support Release (STEP 7 V13 SP1)
   //02.00.01 02.03.2017 Siemens Industry Online Support Release (STEP 7 V14)
   //=============================================================================
   // check parameter
   IF #tmLag1 <= 0 OR #tmLag2 <= 0 OR #tmLag3 <= 0 THEN
     #error := TRUE;
     #status := W#16#8001;     // Parameter Error
     #output := #input; //write output data
     #statFback1 := #input; //write static data
     #statFback2 := #input;
     #statFback3 := #input;
     RETURN;
   ELSE
     #error := FALSE;
     #status := W#16#0000;     // no error
   END_IF;

   IF #reset THEN //complete restart routine

     #output := #input;//write output data
     #statFback1 := #input;//write static data
     #statFback2 := #input;
     #statFback3 := #input;

   ELSE //cycle mode routine

     #tempCycleR  := #cycle*1000; //transform data type
     #tempTmLag1R := #tmLag1*1000;
     #tempTmLag2R := #tmLag2*1000;
     #tempTmLag3R := #tmLag3*1000;

     IF #tempCycleR * 0.5 > #tempTmLag1R THEN //limit TM_LAG1
       #tempTmLag1R := #tempCycleR * 0.5;
     END_IF;

     IF #tempCycleR * 0.5 > #tempTmLag2R THEN //limit TM_LAG2
       #tempTmLag2R := #tempCycleR * 0.5;
     END_IF;

     IF #tempCycleR * 0.5 > #tempTmLag3R THEN //limit TM_LAG2
       #tempTmLag3R := #tempCycleR * 0.5;
     END_IF;

     //1. first order lag algorithm
     #tempHvar     := #tempCycleR / (#tempTmLag1R * 2.0); 
     #tempHvar     := (#gain * (#input + #disturb) - #statFback1) * #tempHvar / (#tempHvar + 1.0);
     #tempOutvNew  := #tempHvar + #statFback1;
     #statFback1  := #tempHvar * 2.0 + #statFback1;

     //2. first order lag algorithm
     #tempHvar     := #tempCycleR / (#tempTmLag2R * 2.0); 
     #tempHvar     := ((#tempOutvNew - #statFback2) * #tempHvar) / (#tempHvar + 1.0);
     #tempOutvNew  := #tempHvar + #statFback2;
     #statFback2  := #tempHvar * 2.0 + #statFback2;

     //3. first order lag algorithm
     #tempHvar     := #tempCycleR / (#tempTmLag3R * 2.0); 
     #tempHvar     := ((#tempOutvNew - #statFback3) * #tempHvar) / (#tempHvar + 1.0);
     #tempOutvNew  := #tempHvar + #statFback3;
     #statFback3  := #tempHvar * 2.0 + #statFback3;

     #output := #tempOutvNew; //write output

   END_IF;
END_FUNCTION_BLOCK

FUNCTION "Byte数组_to_INT" : Void   // FC52, SCL
{ S7_Optimized_Access := 'TRUE' }
VERSION : 0.1
// stored: AutoNumber false, IsIECCheckEnabled false, SetENOAutomatically false, UDAEnableTagReadback false
   VAR_INPUT
      byte数组 : Array[*] of Byte;
      起始偏置 : Int;   // 从数组的第偏置位开始
   END_VAR
   VAR_OUTPUT
      "INT" : Int;
   END_VAR
   VAR_TEMP
      temp_int : Int;
   END_VAR
BEGIN

   #temp_int:=BYTE_TO_INT(#byte数组[#起始偏置]);
   #INT := SHL(IN := #temp_int, N := 8) + #byte数组[#起始偏置 + 1];
END_FUNCTION

FUNCTION "LBitToDword" : Void   // FC231, SCL
TITLE = LBitToDWord
{ S7_Optimized_Access := 'FALSE' }
AUTHOR : Willaim
FAMILY : Control
VERSION : 0.1
// //============================================================================================
// //2017-04-21 15h49
// //Handles the conversion from bits to one DWord.
// //============================================================================================
// stored: AutoNumber false, IsIECCheckEnabled false, SetENOAutomatically false, UDAEnableTagReadback false
   VAR_INPUT
      I_Input0 : Bool;
      I_Input1 : Bool;
      I_Input2 : Bool;
      I_Input3 : Bool;
      I_Input4 : Bool;
      I_Input5 : Bool;
      I_Input6 : Bool;
      I_Input7 : Bool;
      I_Input8 : Bool;
      I_Input9 : Bool;
      I_Input10 : Bool;
      I_Input11 : Bool;
      I_Input12 : Bool;
      I_Input13 : Bool;
      I_Input14 : Bool;
      I_Input15 : Bool;
      I_Input16 : Bool;
      I_Input17 : Bool;
      I_Input18 : Bool;
      I_Input19 : Bool;
      I_Input20 : Bool;
      I_Input21 : Bool;
      I_Input22 : Bool;
      I_Input23 : Bool;
      I_Input24 : Bool;
      I_Input25 : Bool;
      I_Input26 : Bool;
      I_Input27 : Bool;
      I_Input28 : Bool;
      I_Input29 : Bool;
      I_Input30 : Bool;
      I_Input31 : Bool;
   END_VAR
   VAR_OUTPUT
      O_DWordOut : DWord;
   END_VAR
   VAR_TEMP
      TempInputBit : Array[0..31] of Bool;
      TempDWord AT TempInputBit : DWord;
   END_VAR
BEGIN
   //============================================================================================
   //2017-04-21 15h49
   //Handles the conversion from bits to one DWord.
   //============================================================================================

   //**** 1 - Inputs ****  Move Bit to temporary bit.
   #TempInputBit[24] := #I_Input0;
   #TempInputBit[25] := #I_Input1;
   #TempInputBit[26] := #I_Input2;
   #TempInputBit[27] := #I_Input3;
   #TempInputBit[28] := #I_Input4;
   #TempInputBit[29] := #I_Input5;
   #TempInputBit[30] := #I_Input6;
   #TempInputBit[31] := #I_Input7;

   #TempInputBit[16] := #I_Input8;
   #TempInputBit[17] := #I_Input9;
   #TempInputBit[18] := #I_Input10;
   #TempInputBit[19] := #I_Input11;
   #TempInputBit[20] := #I_Input12;
   #TempInputBit[21] := #I_Input13;
   #TempInputBit[22] := #I_Input14;
   #TempInputBit[23] := #I_Input15;

   #TempInputBit[8]  := #I_Input16;
   #TempInputBit[9]  := #I_Input17;
   #TempInputBit[10] := #I_Input18;
   #TempInputBit[11] := #I_Input19;
   #TempInputBit[12] := #I_Input20;
   #TempInputBit[13] := #I_Input21;
   #TempInputBit[14] := #I_Input22;
   #TempInputBit[15] := #I_Input23;

   #TempInputBit[0]  := #I_Input24;
   #TempInputBit[1]  := #I_Input25;
   #TempInputBit[2]  := #I_Input26;
   #TempInputBit[3]  := #I_Input27;
   #TempInputBit[4]  := #I_Input28;
   #TempInputBit[5]  := #I_Input29;
   #TempInputBit[6]  := #I_Input30;
   #TempInputBit[7]  := #I_Input31;

   //**** 8 - Outputs **** Move the temporary DWord to the output DWord
   #O_DWordOut := #TempDWord;
END_FUNCTION

FUNCTION "LBitToWord" : Void   // FC232, SCL
TITLE = LBitToWord
{ S7_Optimized_Access := 'FALSE' }
AUTHOR : William
FAMILY : Control
VERSION : 0.1
// //============================================================================================
// //2017-04-21 15h49
// //Moves the 16 input bits to one output integer.
// //============================================================================================
// stored: AutoNumber false, IsIECCheckEnabled false, SetENOAutomatically false, UDAEnableTagReadback false
   VAR_INPUT
      I_Input0 : Bool;
      I_Input1 : Bool;
      I_Input2 : Bool;
      I_Input3 : Bool;
      I_Input4 : Bool;
      I_Input5 : Bool;
      I_Input6 : Bool;
      I_Input7 : Bool;
      I_Input8 : Bool;
      I_Input9 : Bool;
      I_Input10 : Bool;
      I_Input11 : Bool;
      I_Input12 : Bool;
      I_Input13 : Bool;
      I_Input14 : Bool;
      I_Input15 : Bool;
   END_VAR
   VAR_OUTPUT
      O_WordOut : Word;   // Output Word format
   END_VAR
   VAR_TEMP
      TempInputBit : Array[0..15] of Bool;
      TempWord AT TempInputBit : Word;
   END_VAR
BEGIN
   //============================================================================================
   //2017-04-21 15h49
   //Moves the 16 input bits to one output integer.
   //============================================================================================

   //**** 1 - Inputs ****  Move Bit to temporary bit.
   #TempInputBit[8] := #I_Input0;
   #TempInputBit[9] := #I_Input1;
   #TempInputBit[10] := #I_Input2;
   #TempInputBit[11] := #I_Input3;
   #TempInputBit[12] := #I_Input4;
   #TempInputBit[13] := #I_Input5;
   #TempInputBit[14] := #I_Input6;
   #TempInputBit[15] := #I_Input7;

   #TempInputBit[0] := #I_Input8;
   #TempInputBit[1] := #I_Input9;
   #TempInputBit[2] := #I_Input10;
   #TempInputBit[3] := #I_Input11;
   #TempInputBit[4] := #I_Input12;
   #TempInputBit[5] := #I_Input13;
   #TempInputBit[6] := #I_Input14;
   #TempInputBit[7] := #I_Input15;


   //**** 8 - Outputs **** Move the temporary Word to the output Word
   #O_WordOut := #TempWord;
END_FUNCTION

FUNCTION "Real_to_Time" : Void   // FC46, SCL
{ S7_Optimized_Access := 'TRUE' }
VERSION : 0.1
// stored: AutoNumber true, IsIECCheckEnabled false, SetENOAutomatically false, UDAEnableTagReadback false
   VAR_INPUT
      "Real" : Real;   // 单位：秒
   END_VAR
   VAR_OUTPUT
      "Time" : Time;
   END_VAR
   VAR_TEMP
      Dint_Temp : DInt;
   END_VAR
BEGIN
   #Time := DINT_TO_TIME(REAL_TO_DINT(#Real * 1000.0));
END_FUNCTION

FUNCTION "数组最大平均值" : Void   // FC34, SCL
{ S7_Optimized_Access := 'TRUE' }
VERSION : 0.1
// stored: AutoNumber true, IsIECCheckEnabled false, SetENOAutomatically false, UDAEnableTagReadback false
   VAR_INPUT
      输入数组 : Variant;   // 输入的数组，这里是泛型类型(P#这种数组指针写法)
   END_VAR
   VAR_OUTPUT
      max_out : Variant;   // 最大值输出（无效输出）
      最大值在数组内的索引 : DInt;   // 最大值索引（由于输入数组的类型不确定，无法给出最大值，只能得到数组最大值的索引，其他地方通过索引去访问）
      报错消息 : String;   // 报错消息
      平均值 : LReal;   // 平均值
   END_VAR
   VAR_TEMP
      arr_length : DInt;   // 传入数组的长度值
      i : DInt;   // 循环次数
      arr_int_temp : Array[0..#max_length] of Int;   // 把输入的数组暂存变量int
      max_number_temp_int : Int;   // 最大值暂存int
      arr_real_temp : Array[0..#max_length] of Real;   // 把输入的数组暂存变量real
      max_number_temp_real : Real;   // 最大值的暂存real
      max_index_temp : DInt;   // 最大值的索引暂存
      sum : LReal;   // 数组和
   END_VAR
   VAR CONSTANT
      max_length : DInt := 201;   // 所能处理的最大数组长度，可修改
   END_VAR
BEGIN
   //本程序的数组输入索引是必须从0开始
   IF IS_ARRAY(#输入数组) THEN //判断是否是数组

       #arr_length := UDINT_TO_DINT(CountOfElements(#输入数组)); //找到数组的长度，函数返回值类型是UDINT,要转成DINT

       IF #arr_length < #max_length THEN //如果输入的数组的长度小于设定的最大长度 则进行以下判断

           //**************************判断数组是整数进行计算***************************************

           IF TypeOfElements(#输入数组) = Int THEN //判断输入数组的类型

               VariantGet(SRC := #输入数组,

                          DST => #arr_int_temp);

               #max_number_temp_int := #arr_int_temp[0]; //把索引为0的数认为是最大值

               #max_index_temp := 0; //把0索引存起来

               FOR #i := 0 TO #max_length - 1 DO //循环 从最小索引开始，到最大索引结束

                   IF #max_number_temp_int < #arr_int_temp[#i] THEN //如果最大值小于后面索引的值

                       #max_number_temp_int := #arr_int_temp[#i]; //则把后面索引的值存入最大值变量里

                       #max_index_temp := #i; //再把索引存起来

                   END_IF;

                   #sum := #sum + #arr_int_temp[#i];

               END_FOR;

               VariantPut(SRC := #max_number_temp_int,

                          DST := #max_out); //把最大值输出 int

               #最大值在数组内的索引 := #max_index_temp; //把最大值的索引输出

               #平均值 := #sum / #arr_length;

               //*******************************如果数组是浮点进行计算*********************************

           ELSIF TypeOfElements(#输入数组) = Real THEN //判断输入数组的类型

               VariantGet(SRC := #输入数组,

                          DST => #arr_real_temp); //把输入的数组传入到内部数组进行处理

               #max_number_temp_real := #arr_real_temp[0]; //把索引为0的数认为是最大值

               #max_index_temp := 0; //把0索引存起来

               FOR #i := 0 TO #max_length - 1 DO //循环 从最小索引开始，到最大索引结束

                   IF #max_number_temp_real < #arr_real_temp[#i] THEN //如果最大值小于后面索引的值

                       #max_number_temp_real := #arr_real_temp[#i]; //则把后面索引的值存入最大值变量里

                       #max_index_temp := #i; //再把索引存起来

                   END_IF;

                   #sum := #sum + #arr_real_temp[#i];

               END_FOR;

               VariantPut(SRC := #max_number_temp_real,

                          DST := #max_out); //把最大值输出 real

               #最大值在数组内的索引 := #max_index_temp; //把最大值的索引输出

               #平均值 := #sum / #arr_length;

           END_IF;

       ELSE

           #报错消息 := 'fault'; //如果输入的数组长度超过200个，那就报错

       END_IF;

   END_IF;
END_FUNCTION

FUNCTION "相减日期和时间" : Void   // FC3108, STL
TITLE = Data_And_Time减法运算
{ S7_Optimized_Access := 'FALSE' }
VERSION : 0.1
// stored: AutoNumber true, UDAEnableTagReadback false
   VAR_INPUT
      被减时间 : Pointer;   // 被减时间(Data_And_Time类型)
      减数时间 : Pointer;   // 减数(Data_And_Time类型)
      TimeOver : Bool;   // 时间到达
   END_VAR
   VAR_OUTPUT
      剩余时间 : Pointer;   // 剩余时间(Data_And_Time类型)
   END_VAR
   VAR_TEMP
      Minu : Struct
         year : Int;   // 年
         mouth : Int;   // 月
         day : Int;   // 日
         hour : Int;   // 时
         min : Int;   // 分
         sec : Int;   // 秒
      END_STRUCT;
      Sub : Struct
         year : Int;   // 年
         mouth : Int;   // 月
         day : Int;   // 日
         hour : Int;   // 时
         min : Int;   // 分
         sec : Int;   // 秒
      END_STRUCT;
      Res : Struct
         year : Int;   // 年
         mouth : Int;   // 月
         day : Int;   // 日
         hour : Int;   // 时
         min : Int;   // 分
         sec : Int;   // 秒
      END_STRUCT;
      MinuDB : Int;
      SubDB : Int;
      ResDB : Int;
      temp1 : Byte;
      temp2 : Byte;
      temp3 : Byte;
      temp4 : Byte;
      temp5 : Byte;
      temp6 : Byte;
      temp7 : Byte;
      temp8 : Byte;
      temp9 : Byte;
      temp10 : Byte;
      temp11 : Byte;
      temp12 : Byte;
      temp13 : Byte;
      temp14 : Byte;
      temp15 : Byte;
      temp16 : Byte;
   END_VAR
BEGIN

NETWORK
TITLE = 指针提取
      L     P##被减时间;  //提取被减时间
      LAR1;
      L     P##减数时间;  //提取被时间
      LAR2;

      L     W [AR1, P#0.0];
      T     #MinuDB;
      L     W [AR2, P#0.0];
      T     #SubDB;
      L     W [AR1, P#4.0];
      LAR1;
      L     W [AR2, P#4.0];
      LAR2;

      A     #TimeOver;
      JC    OVER;


NETWORK
TITLE = 被减时间提取，转化为DEC
      OPN   DB [#MinuDB];
      L     DBB [AR1, P#0.0];
      SRW   4;
      L     10;
      *I;
      T     #temp1;
      L     DBB [AR1, P#0.0];
      L     b#16#0f;
      AW;
      L     #temp1;
      +I;
      T     #Minu.year;  // year

      OPN   DB [#MinuDB];
      L     DBB [AR1, P#1.0];
      SRW   4;
      L     10;
      *I;
      T     #temp2;
      L     DBB [AR1, P#1.0];
      L     b#16#0f;
      AW;
      L     #temp2;
      +I;
      T     #Minu.mouth;  // mouth

      OPN   DB [#MinuDB];
      L     DBB [AR1, P#2.0];
      SRW   4;
      L     10;
      *I;
      T     #temp3;
      L     DBB [AR1, P#2.0];
      L     b#16#0f;
      AW;
      L     #temp3;
      +I;
      T     #Minu.day;  // day

      OPN   DB [#MinuDB];
      L     DBB [AR1, P#3.0];
      SRW   4;
      L     10;
      *I;
      T     #temp4;
      L     DBB [AR1, P#3.0];
      L     b#16#0f;
      AW;
      L     #temp4;
      +I;
      T     #Minu.hour;  // hour

      OPN   DB [#MinuDB];
      L     DBB [AR1, P#4.0];
      SRW   4;
      L     10;
      *I;
      T     #temp5;
      L     DBB [AR1, P#4.0];
      L     b#16#0f;
      AW;
      L     #temp5;
      +I;
      T     #Minu.min;  // min

      OPN   DB [#MinuDB];
      L     DBB [AR1, P#5.0];
      SRW   4;
      L     10;
      *I;
      T     #temp6;
      L     DBB [AR1, P#5.0];
      L     b#16#0f;
      AW;
      L     #temp6;
      +I;
      T     #Minu.sec;  // sec


NETWORK
TITLE = 减时间提取，转化为DEC
      OPN   DB [#SubDB];
      L     DBB [AR2, P#0.0];
      SRW   4;
      L     10;
      *I;
      T     #temp7;
      L     DBB [AR2, P#0.0];
      L     b#16#0f;
      AW;
      L     #temp7;
      +I;
      T     #Sub.year;  // year

      OPN   DB [#SubDB];
      L     DBB [AR2, P#1.0];
      SRW   4;
      L     10;
      *I;
      T     #temp8;
      L     DBB [AR2, P#1.0];
      L     b#16#0f;
      AW;
      L     #temp8;
      +I;
      T     #Sub.mouth;  // mouth

      OPN   DB [#SubDB];
      L     DBB [AR2, P#2.0];
      SRW   4;
      L     10;
      *I;
      T     #temp9;
      L     DBB [AR2, P#2.0];
      L     b#16#0f;
      AW;
      L     #temp9;
      +I;
      T     #Sub.day;  // day

      OPN   DB [#SubDB];
      L     DBB [AR2, P#3.0];
      SRW   4;
      L     10;
      *I;
      T     #temp10;
      L     DBB [AR2, P#3.0];
      L     b#16#0f;
      AW;
      L     #temp10;
      +I;
      T     #Sub.hour;  // hour

      OPN   DB [#SubDB];
      L     DBB [AR2, P#4.0];
      SRW   4;
      L     10;
      *I;
      T     #temp11;
      L     DBB [AR2, P#4.0];
      L     b#16#0f;
      AW;
      L     #temp11;
      +I;
      T     #Sub.min;  // min

      OPN   DB [#SubDB];
      L     DBB [AR2, P#5.0];
      SRW   4;
      L     10;
      *I;
      T     #temp12;
      L     DBB [AR2, P#5.0];
      L     b#16#0f;
      AW;
      L     #temp12;
      +I;
      T     #Sub.sec;  // sec


NETWORK
TITLE = 减法运算
      L     #Minu.year;
      L     #Sub.year;
      -I;
      T     #Res.year;

      L     #Minu.mouth;
      L     #Sub.mouth;
      -I;
      T     #Res.mouth;

      L     #Minu.day;
      L     #Sub.day;
      -I;
      T     #Res.day;

      L     #Minu.hour;
      L     #Sub.hour;
      -I;
      T     #Res.hour;

      L     #Minu.min;
      L     #Sub.min;
      -I;
      T     #Res.min;

      L     #Minu.sec;
      L     #Sub.sec;
      -I;
      T     #Res.sec;


NETWORK
TITLE = 被减数小于减数，向高位借1
      A(;
      L     #Res.sec;
      L     0;
      <I;
      );
      JCN   _001;
      L     #Res.sec;
      L     60;
      +I;
      T     #Res.sec;
      L     #Res.min;
      L     1;
      -I;
      T     #Res.min;
_001: A(;
      L     #Res.min;
      L     0;
      <I;
      );
      JCN   _002;
      L     #Res.min;
      L     60;
      +I;
      T     #Res.min;
      L     #Res.hour;
      L     1;
      -I;
      T     #Res.hour;
_002: A(;
      L     #Res.hour;
      L     0;
      <I;
      );
      JCN   _003;
      L     #Res.hour;
      L     24;
      +I;
      T     #Res.hour;
      L     #Res.day;
      L     1;
      -I;
      T     #Res.day;
_003: A(;
      L     #Res.day;
      L     0;
      <I;
      );
      JCN   _004;
      L     #Res.day;
      L     30;
      +I;
      T     #Res.day;
      L     #Res.mouth;
      L     1;
      -I;
      T     #Res.mouth;
_004: A(;
      L     #Res.mouth;
      L     0;
      <I;
      );
      JCN   _111;
      L     #Res.mouth;
      L     12;
      +I;
      T     #Res.mouth;
      L     #Res.year;
      L     1;
      -I;
      T     #Res.year;
_111: NOP   0;
      JU    Resi;

NETWORK
TITLE = time over
OVER: L     0;
      T     #Res.year;
      T     #Res.mouth;
      T     #Res.day;
      T     #Res.hour;
      T     #Res.min;
      T     #Res.sec;


NETWORK
TITLE = 差值赋值到剩余时间
Resi: L     P##剩余时间;  //提取剩余时间
      LAR1;
      L     W [AR1, P#0.0];
      T     #ResDB;
      L     W [AR1, P#4.0];
      LAR1;

      OPN   DB [#ResDB];
      L     #Res.year;
      T     DBB [AR1, P#0.0];
      L     #Res.mouth;
      T     DBB [AR1, P#1.0];
      L     #Res.day;
      T     DBB [AR1, P#2.0];
      L     #Res.hour;
      T     DBB [AR1, P#3.0];
      L     #Res.min;
      T     DBB [AR1, P#4.0];
      L     #Res.sec;
      T     DBB [AR1, P#5.0];



NETWORK
TITLE = RLO
      SET;
      SAVE;

END_FUNCTION

FUNCTION "随机生成数" : Void   // FC39, SCL
{ S7_Optimized_Access := 'TRUE' }
VERSION : 0.1
// stored: AutoNumber true, IsIECCheckEnabled false, SetENOAutomatically false, UDAEnableTagReadback false
   VAR_INPUT
      最小生成数 : Real;
      偏置 : Real;
      数据类型 : Bool;   // 0为实数，1为整数
   END_VAR
   VAR_OUTPUT
      随机数 : Real;
   END_VAR
BEGIN
   IF #数据类型 THEN
       #随机数 := REAL_TO_DINT(INT_TO_REAL("Clock_Byte") / 255 * #偏置 + #最小生成数);
   ELSE
       #随机数 := INT_TO_REAL("Clock_Byte") / 255 * #偏置 + #最小生成数;
   END_IF;
END_FUNCTION

FUNCTION_BLOCK "TX通讯心跳"   // FB61, SCL
{ S7_Optimized_Access := 'TRUE' }
VERSION : 0.1
// stored: AutoNumber true, IsIECCheckEnabled false, IsRetainMemResEnabled false, MemoryReserve 100, SetENOAutomatically false, UDAEnableTagReadback false
   VAR_INPUT
      XH信号不同超时报警 : Real := 120.0;   // SB设备写读与创造写对比,如果不同超时,即判断报警
      XH信号相同超时报警 : Real := 120.0;   // SB设备写读与创造写对比,如果相同超时,即判断报警
      MC脉冲切换时间 : Real := 20.0;   // 给写信号+1,创造不同，10秒切换一次
   END_VAR
   VAR_OUTPUT
      设备未通信报警 : Bool;
   END_VAR
   VAR_IN_OUT
      SB设备写读 : Real;
      SB设备写 : Real;
      SB设备检测写 : Real;
   END_VAR
   VAR
      TON1 { S7_SetPoint := 'True'} : TON_TIME;
      TON1ET { S7_SetPoint := 'True'} : Time;
      TON2 : TON_TIME;
      TON2ET { S7_SetPoint := 'True'} : Time;
      LS设备通延辅助1 { S7_SetPoint := 'True'} : Bool;
      LS设备通延辅助2 : Bool;
      LS通信脉冲读1 : Bool;
      LS通信脉冲读2 : Bool;
      LS设备读温比较 : Real;
      T1S : TON_TIME;
      YC1 { S7_SetPoint := 'True'} : Real;
   END_VAR
   VAR_TEMP
      "m" : Int;
   END_VAR
BEGIN
   IF "FirstScan" THEN
       RESET_TIMER(#TON1);
       RESET_TIMER(#TON2);
       #LS设备通延辅助1 := 0;
       #LS设备通延辅助2 := 0;
   END_IF;

   IF #T1S.Q AND #YC1<#MC脉冲切换时间 THEN
       #YC1 := #YC1 + 1;
   END_IF;

   IF #YC1 >= #MC脉冲切换时间 THEN
       #YC1 := 0;
   END_IF;

   IF #YC1 <= (#MC脉冲切换时间 - 10) THEN

       #LS通信脉冲读1 := 1;
       #LS通信脉冲读2 := 0;
   ELSE
       #LS通信脉冲读1 := 0;
       #LS通信脉冲读2 := 1;
   END_IF;

   IF #LS通信脉冲读1 THEN
       //冷水
       #LS设备读温比较 := #SB设备写读;
       #SB设备检测写 := #SB设备写 + 0.1;
       #TON1(IN := (ABS(#LS设备读温比较) <> ABS(#SB设备检测写)),
             PT := DINT_TO_TIME(REAL_TO_DINT(#XH信号不同超时报警 * 1000.0)),
             Q => #LS设备通延辅助1,
             ET => #TON1ET);

      #TON2(IN := (ABS(#LS设备读温比较) = ABS(#SB设备检测写)),
             PT := DINT_TO_TIME(REAL_TO_DINT(#XH信号相同超时报警 * 1000.0)),
             Q => #LS设备通延辅助2,
             ET => #TON2ET);

   END_IF;

   IF #LS通信脉冲读2 THEN
       #SB设备检测写 := #SB设备写;
   END_IF;

   IF #LS设备通延辅助1 OR #LS设备通延辅助2  THEN
       #设备未通信报警 := 1;
   ELSE
       #设备未通信报警 := 0;
   END_IF;

   #T1S(IN := NOT #T1S.Q,
       PT := T#1S);
END_FUNCTION_BLOCK

FUNCTION_BLOCK "上升沿"   // FB59, SCL
{ S7_Optimized_Access := 'TRUE' }
VERSION : 0.1
// stored: AutoNumber true, IsIECCheckEnabled false, IsRetainMemResEnabled false, MemoryReserve 100, SetENOAutomatically false, UDAEnableTagReadback false
   VAR_INPUT
      IN : Bool;
   END_VAR
   VAR_IN_OUT
      Q : Bool;
      State : Bool;
   END_VAR
   VAR
      RT1 { S7_SetPoint := 'True'} : R_TRIG;
   END_VAR
BEGIN
   #RT1(CLK := #IN);
   IF #RT1.Q THEN
       #Q := 1;
   END_IF;
   #State := #RT1.Stat_Bit;
END_FUNCTION_BLOCK

FUNCTION_BLOCK "单元模式"   // FB81, SCL
{ S7_Optimized_Access := 'TRUE' }
VERSION : 0.1
// stored: AutoNumber true, IsIECCheckEnabled false, IsRetainMemResEnabled false, MemoryReserve 100, SetENOAutomatically false, UDAEnableTagReadback false
   VAR
      第一动作中 : Bool;
      第二动作中 : Bool;
      动作信号 : Bool;
      estop : Bool;
      动作按钮 : Bool;
      动作超时 : Bool;
      动作条件 : Bool;
      动作到位 : Bool;
      动作输出 : Bool;
      手动模式 : Bool;
      自动模式 : Bool;
      超时 : TON_TIME;
      故障复位 : Bool;
      反馈信号 : Bool;
   END_VAR
BEGIN
   #动作信号 := #第一动作中 OR #第二动作中;
   #动作条件 := NOT #estop AND NOT #动作超时;
   IF ((#自动模式 AND #动作信号) OR (#手动模式 AND #动作按钮) OR #动作输出)
       AND #动作条件
       AND NOT #动作到位 THEN
       #动作输出 := 1;
   ELSE
       #动作输出 := 0;
   END_IF;

   #动作到位 := #反馈信号;

   #超时(IN:=(#动作输出 AND NOT #动作到位),
       PT:=T#5S);

   #动作超时 := #超时.Q OR (#动作超时 AND NOT #故障复位);
END_FUNCTION_BLOCK

FUNCTION_BLOCK "启停模式"   // FB51, SCL
{ S7_Optimized_Access := 'TRUE' }
VERSION : 0.1
// stored: AutoNumber true, IsIECCheckEnabled false, IsRetainMemResEnabled false, MemoryReserve 100, SetENOAutomatically false, UDAEnableTagReadback false
   VAR
      Start : Bool;
      Stop : Bool;
      RUN : Bool;
   END_VAR
BEGIN
   #RUN := (#Start OR #RUN) AND NOT #Stop;
END_FUNCTION_BLOCK

FUNCTION_BLOCK "抖动模式"   // FB44, SCL
{ S7_Optimized_Access := 'TRUE' }
VERSION : 0.1
// stored: AutoNumber true, IsIECCheckEnabled false, IsRetainMemResEnabled false, MemoryReserve 100, SetENOAutomatically false, UDAEnableTagReadback false
   VAR_INPUT
      ONY : Time := T#3S;
      OFY : Time := T#2S;
   END_VAR
   VAR_IN_OUT
      IN : Bool;
      OUT : Bool;
   END_VAR
   VAR
      TON { ExternalAccessible := 'False'; ExternalVisible := 'False'; ExternalWritable := 'False'} : TON_TIME;
      TOF { ExternalAccessible := 'False'; ExternalVisible := 'False'; ExternalWritable := 'False'} : TOF_TIME;
   END_VAR
BEGIN

   #TON(IN:=#IN,
        PT:=#ONY);
   #TOF(IN := #IN,
        PT := #OFY);
   #OUT:=#TON.Q OR (#TOF.Q AND #OUT) ;
END_FUNCTION_BLOCK

FUNCTION_BLOCK "斜坡函数发生器"   // FB85, SCL
{ S7_Optimized_Access := 'TRUE' }
VERSION : 0.1
// stored: AutoNumber true, IsIECCheckEnabled false, IsRetainMemResEnabled false, MemoryReserve 100, SetENOAutomatically false, UDAEnableTagReadback false
   VAR_INPUT
      输入 : Real;
      斜坡激活 : Bool;   // 0：直接输出 1：斜坡输出
      上升斜率 : Real := 1.0;   // 斜坡上升增量值 （单位值/秒）
      下降斜率 : Real := 1.0;   // 斜坡下降增量值 （ 单位值/秒）
      输出上限 : Real := 100.0;
      输出下限 : Real := 0.0;
   END_VAR
   VAR_OUTPUT
      输出 : Real;
   END_VAR
BEGIN

   //可用于电机的速度给定以实现平滑升/降速；重要的调节阀门设定，进行平滑过度，防止水锤及工艺扰动等现象
   //在循环中断OB30中调用该FB块，OB30循环时间设置为100ms。
   //如果上升斜率设置为1/s，输入则上升斜坡将持续10s（设定值从0增加至10）。
   //公式：Y=Y+A。

   IF NOT #斜坡激活 THEN
       //直接输出
       #输出 := #输入;
   ELSE
       //斜坡输出
       IF #输入 > #输出 THEN
           //斜坡上升
           #输出 := #输出 + #上升斜率 / 10.0;
       END_IF;
       IF #输入 < #输出 THEN
           //斜坡下降
           #输出 := #输出 - #下降斜率 / 10.0;
       END_IF;
   END_IF;


   //输出限幅
   IF #输出 > #输出上限 THEN
       #输出 := #输出上限;
   END_IF;
   IF #输出 < #输出下限 THEN
       #输出 := #输出下限;
   END_IF;
END_FUNCTION_BLOCK

FUNCTION_BLOCK "时间累计"   // FB66, SCL
{ S7_Optimized_Access := 'TRUE' }
VERSION : 0.1
// stored: AutoNumber true, IsIECCheckEnabled false, IsRetainMemResEnabled false, MemoryReserve 100, SetENOAutomatically false, UDAEnableTagReadback false
   VAR_INPUT
      start : Bool;
      reset : Bool;
   END_VAR
   VAR_OUTPUT
      h : Int;
      "m" : Int;
      s : Int;
   END_VAR
   VAR
      T1S : TON_TIME;
   END_VAR
BEGIN

   IF #start AND #T1S.Q THEN
       #s := #s + 1;
   END_IF;
   IF #reset THEN
       #h := 0;
       #m := 0;
       #s := 0;
   END_IF;
   IF #s >= 60 THEN
       #m := #m + 1;
       #s := 0;
   END_IF;

   IF #m >= 60 THEN
       #h := #h + 1;
       #m := 0;
   END_IF;

   #T1S(IN := NOT #T1S.Q,
        PT := T#1S);
END_FUNCTION_BLOCK

FUNCTION_BLOCK "步模式"   // FB60, SCL
{ S7_Optimized_Access := 'TRUE' }
VERSION : 0.1
// stored: AutoNumber true, IsIECCheckEnabled false, IsRetainMemResEnabled false, MemoryReserve 100, SetENOAutomatically false, UDAEnableTagReadback false
   VAR_INPUT
      FK : Bool;   // 动作反馈
   END_VAR
   VAR_IN_OUT
      IN : Bool;   // 进入步段条件
      RUN : Bool;   // 动作运行,运行完后就关闭,一般接TON
      DONE : Bool;   // 动作完成,一般是一个标注位
      OVER : Bool;   // 步段完成,运行完之后继续开状态
   END_VAR
BEGIN
   #OVER := #IN AND (#DONE OR #OVER);
   #RUN := #IN AND NOT #OVER ;
   #DONE := #RUN AND #FK;
END_FUNCTION_BLOCK

FUNCTION_BLOCK "步段延迟"   // FB65, SCL
{ S7_Optimized_Access := 'TRUE' }
VERSION : 0.1
// stored: AutoNumber true, IsIECCheckEnabled false, IsRetainMemResEnabled false, MemoryReserve 100, SetENOAutomatically false, UDAEnableTagReadback false
   VAR_INPUT
      YC延迟设定时间 : Real := 50.0;   // 设定延迟时间
   END_VAR
   VAR_IN_OUT
      "AND" : Bool;   // 延迟的条件
      Q : Bool;   // 延迟时间到达后执行的动作
      YX运行时间 : Real;   // 显示时钟时间
   END_VAR
   VAR
      T1S : TON_TIME;   // 1秒脉冲
   END_VAR
BEGIN
   IF #T1S.Q AND #YX运行时间 < #YC延迟设定时间 AND #AND THEN
       #YX运行时间 := #YX运行时间 + 1;
   END_IF;

   IF #YX运行时间 >= #YC延迟设定时间 THEN
       #Q := 1;
   END_IF;

   (* IF NOT #AND THEN
       #YX运行时间 := 0;
       #Q := 0;
   END_IF; *)

   #T1S(IN := NOT #T1S.Q,
          PT := T#1S);
END_FUNCTION_BLOCK

FUNCTION_BLOCK "步段延迟案例"   // FB70, SCL
{ S7_Optimized_Access := 'TRUE' }
VERSION : 0.1
// stored: AutoNumber true, IsIECCheckEnabled false, IsRetainMemResEnabled false, MemoryReserve 100, SetENOAutomatically false, UDAEnableTagReadback false
   VAR_IN_OUT
      BD步段运行 : Int;
      BD步段设定 : Int;
   END_VAR
   VAR
      STEP1 { S7_SetPoint := 'True'} : "步段延迟";
      STEP2 { S7_SetPoint := 'True'} : "步段延迟";
      STEP3 { S7_SetPoint := 'True'} : "步段延迟";
   END_VAR
BEGIN
   CASE #BD步段运行 OF
       1:
           #STEP1.AND := #BD步段运行 = 1;
           #STEP1(YC延迟设定时间:=30.0);


           IF #STEP1.Q THEN
               #BD步段运行 := 2;
           END_IF;
           ;
       2:
           #STEP2.AND := #BD步段运行 = 2;
           #STEP2(YC延迟设定时间 := 30.0);
           IF #STEP2.Q THEN


               #BD步段运行 := 3;
           END_IF;
           ;
       3:
           #STEP3.AND := #BD步段运行 = 3;
           #STEP3(YC延迟设定时间 := 30.0);
           IF #STEP3.Q THEN
               #BD步段运行 := 1;
           END_IF;

   END_CASE;


   IF #BD步段设定 <> #BD步段运行 THEN
       #STEP1.YX运行时间 := 0;
       #STEP2.YX运行时间 := 0;
       #STEP3.YX运行时间 := 0;
       #STEP1.Q := 0;
       #STEP2.Q := 0;
       #STEP3.Q := 0;
       #BD步段设定 := #BD步段运行;
   END_IF;
END_FUNCTION_BLOCK

FUNCTION_BLOCK "沿"   // FB67, LAD
{ S7_Optimized_Access := 'TRUE' }
VERSION : 0.1
// stored: AutoNumber true, IsIECCheckEnabled false, IsRetainMemResEnabled false, MemoryReserve 100, SetENOAutomatically false, UDAEnableTagReadback false
   VAR_INPUT
      IN : Bool;
   END_VAR
   VAR_OUTPUT
      Q : Bool;
   END_VAR
   VAR
      U_1 : Bool;
      L_1 : Bool;
   END_VAR
BEGIN

REGION Network 1 (SCL)
   IF #IN AND NOT #U_1 THEN

       #Q := 1;

   END_IF;

   #U_1 := #IN;
END_REGION
END_FUNCTION_BLOCK

FUNCTION_BLOCK "状态模式"   // FB84, SCL
{ S7_Optimized_Access := 'TRUE' }
VERSION : 0.1
// stored: AutoNumber true, IsIECCheckEnabled false, IsRetainMemResEnabled false, MemoryReserve 100, SetENOAutomatically false, UDAEnableTagReadback false
   VAR
      phaseloss : Bool;
      powerfault : Bool;
      faultreset : Bool;
      sb_start : Bool;
      sb_stop : Bool;
      motor : Bool;
   END_VAR
BEGIN
   #powerfault := #phaseloss OR (#powerfault AND NOT #faultreset);

   #motor := (#sb_start OR #sb_stop) AND NOT #sb_stop AND NOT #powerfault;
END_FUNCTION_BLOCK

FUNCTION_BLOCK "脉冲模式"   // FB39, SCL
{ S7_Optimized_Access := 'TRUE' }
VERSION : 0.1
// stored: AutoNumber true, IsIECCheckEnabled false, IsRetainMemResEnabled false, MemoryReserve 100, SetENOAutomatically false, UDAEnableTagReadback false
   VAR_IN_OUT
      QD : Bool;
      ST1 : Bool;
      ST2 : Bool;
      ST3 : Bool;
   END_VAR
   VAR
      TON1 : TON_TIME;
   END_VAR
BEGIN

   (* #BT1F := DINT_TO_TIME(REAL_TO_DINT(#BT1 * 1000.0));
   #BT2F := DINT_TO_TIME(REAL_TO_DINT(#BT1 * 1000.0)) + DINT_TO_TIME(REAL_TO_DINT(#BT2 * 1000.0));
   #BT3F := DINT_TO_TIME(REAL_TO_DINT(#BT1 * 1000.0)) + DINT_TO_TIME(REAL_TO_DINT(#BT2 * 1000.0)) + DINT_TO_TIME(REAL_TO_DINT(#BT3 * 1000.0));
   #BTAF := DINT_TO_TIME(REAL_TO_DINT(#BT1 * 1000.0)) + DINT_TO_TIME(REAL_TO_DINT(#BT2 * 1000.0)) + DINT_TO_TIME(REAL_TO_DINT(#BT3 * 1000.0)) + T#20S;
   *)
   #ST1 := 0;
   #ST2 := 0;
   #ST3 := 0;
   #QD := 0;


   IF #QD  THEN
       #TON1(IN := NOT #TON1.Q,
             PT := T#50S);

       IF #TON1.ET > T#10S THEN
               #ST1 := 1;
           END_IF;

       IF #TON1.ET >T#20S THEN
           #ST2 := 1;
       END_IF;

       IF #TON1.ET >T#30S THEN
           #ST3 := 1;
       END_IF;

       IF #TON1.ET > T#40S THEN
           #QD := 0;

       END_IF;

   END_IF;
END_FUNCTION_BLOCK

FUNCTION_BLOCK "自保持模式"   // FB83, SCL
{ S7_Optimized_Access := 'TRUE' }
VERSION : 0.1
// stored: AutoNumber true, IsIECCheckEnabled false, IsRetainMemResEnabled false, MemoryReserve 100, SetENOAutomatically false, UDAEnableTagReadback false
   VAR
      dooropened : Bool;
      homed : Bool;
      selfcheckmeet : Bool;
      sb_start : Bool;
      sb_stop : Bool;
      light : Bool;
   END_VAR
BEGIN
   #selfcheckmeet := (#dooropened AND #homed) OR #selfcheckmeet;

   IF NOT #selfcheckmeet THEN
       RETURN;
   END_IF;

   #light := (#sb_start OR #light) AND NOT #sb_stop;
END_FUNCTION_BLOCK

FUNCTION_BLOCK "自动流程"   // FB82, SCL
{ S7_Optimized_Access := 'TRUE' }
VERSION : 0.1
// stored: AutoNumber true, IsIECCheckEnabled false, IsRetainMemResEnabled false, MemoryReserve 100, SetENOAutomatically false, UDAEnableTagReadback false
   VAR
      execute : Bool;
      stepmode : Bool;
      stepsignal : Bool;
      stepsignalrise : Bool;
      stepsignallast : Bool;
      "step" : Int;
      nextstep : Int;
      "1号cmd" : Bool;
      "1号pos" : Bool;
      "1号homecmd" : Bool;
      "1号homepos" : Bool;
      "2号cmd" : Bool;
      "2号pos" : Bool;
      "2号homecmd" : Bool;
      "2号homepos" : Bool;
   END_VAR
BEGIN
   IF #execute THEN
       CASE #step OF
           0:
               #"1号cmd" := 1;
               IF #"1号pos" THEN
                   #"1号cmd" := 0;
                   #nextstep := 10;
               END_IF;
               ;
           10:
               #"2号cmd" := 1;
               IF #"2号pos" THEN
                   #"2号cmd" := 0;
                   #nextstep := 20;
               END_IF;
               ;
           20:
               #"2号homecmd" := 1;
               IF #"2号homepos" THEN
                   #"2号homecmd" := 0;
                   #nextstep := 30;
               END_IF;
               ;
           30:
               #"1号homecmd" := 1;
               IF #"1号homepos" THEN
                   #"1号homecmd" := 0;
                   #nextstep := 40;
               END_IF;
           ELSE
               ;
       END_CASE;

       #stepsignalrise := #stepsignal AND NOT #stepsignallast;
       #stepsignallast := #stepsignal;
       IF NOT #stepmode OR (#stepmode AND #stepsignalrise) THEN
           #step := #nextstep;
       END_IF;
   ELSE
       #step := 0;
   END_IF;
END_FUNCTION_BLOCK

FUNCTION_BLOCK "A1-台达DTC"   // FB33, SCL
{ S7_Optimized_Access := 'TRUE' }
VERSION : 0.1
// stored: AutoNumber true, IsIECCheckEnabled false, IsRetainMemResEnabled false, MemoryReserve 100, SetENOAutomatically false, UDAEnableTagReadback false
   VAR_INPUT
      站号 : UInt;
      触发 : Bool;
      输入模式 : Int;
      输入开关 : Bool;
      A输入设定 : Real;
      输入开度 : Real;
   END_VAR
   VAR_OUTPUT
      结束 : Bool;
      高高报警 : Bool;
      高报警 : Bool;
      低报警 : Bool;
      低低报警 : Bool;
      传感器故障 : Bool;
      输出控制P : Real;
      输出控制I : Real;
      输出控制D : Real;
      输出开度读 : Real;
   END_VAR
   VAR_IN_OUT
      B当前量 : Real;
      输入设定读 : Real;
      输出模式读 : Real;
      高高报设置 : Real;
      高报设置 : Real;
      低报设置 : Real;
      低低报设置 : Real;
      自整定开关 : Bool;
      Modbus_Master_Instance : Modbus_Master;
   END_VAR
   VAR DB_SPECIFIC
      当前指令ID : Int;
      上一次指令ID : Int;
      modbus_data : Struct
         触发 : Bool;
         站号 : UInt;
         模式 : USInt;
         地址 : UDInt;
         数据长度 : UInt;
         完成 : Bool;
         忙碌 : Bool;
         出错 : Bool;
         故障码 : Word;
         数据缓存区 : Array[1..50] of Word;
      END_STRUCT;
      报错代码 : Array[1..20] of Word;
      进温P读 : Int;
      进温I读 : Int;
      进温D读 : Int;
      T1_SV_写 : Int;
      进温AT开关 : Bool;
      进温AT开关_bak : Bool;
      进温AT_写字 : UInt;
      进温AT_读字 : UInt;
      T1_P值比对1 : Int;
      T1_P值比对2 : Int;
      进温启停字 : UInt;
      T1 { S7_SetPoint := 'True'} : TON_TIME;
   END_VAR
   VAR_TEMP
      tm_int : Int;
      tm_real : Real;
   END_VAR
BEGIN
   //程序1

   IF #触发 THEN
       #当前指令ID := 1;
   END_IF;

   #modbus_data.站号 := #站号;

   IF #当前指令ID = 9 THEN
       IF #进温AT_写字 = #进温AT_读字 THEN
           #当前指令ID := 10;
       END_IF;
   END_IF;

   CASE #当前指令ID OF
       1:
           //读取地址44097-44098
           #modbus_data.模式 := 0;
           #modbus_data.地址 := 44097;
           #modbus_data.数据长度 := 2;
       2:
           //读取地址44102
           (* 1005H-4101-44102  默认0   控制方式 0：PID；1：ON/OFF；2：手动；3：PID 过程控制 *)
           #modbus_data.模式 := 0;
           #modbus_data.地址 := 44102;
           #modbus_data.数据长度 := 1;
       3:
           //读取地址44106-44108
           (*  
           1009H-4105-44106  默认476 PB 比例带设定值 1 ~ 9,999, 温度单位为 0.1 度，模拟输入为 1EU
           100AH-4106-44107  默认260 Ti 积分控制常量设定值 0 ~ 9,999
           100BH-4107-44108  默认41 Td 微分控制常量设定值 0 ~ 9,999 *)
           #modbus_data.模式 := 0;
           #modbus_data.地址 := 44106;
           #modbus_data.数据长度 := 3;
       4:
           //读取地址44116
           (* 1013H-4115-44116  默认0   输出 2 输出量读取与写入 单位为 0.1%，写入只在手动控制模式下有效（DTC1000/2000 机种） *)
           #modbus_data.模式 := 0;
           #modbus_data.地址 := 44116;
           #modbus_data.数据长度 := 1;
       5:
           //读取地址12068
           (* 0813H-2067-12068  读写自动调谐状态 自动调谐停止：0（预设），自动调谐开始：1 *)
           #modbus_data.模式 := 0;
           #modbus_data.地址 := 12068;
           #modbus_data.数据长度 := 1;
       6:
           //写入地址44098
           (* 1001H-4097-44098       默认0 "SV" 设定值 温度以 0.1 度为计量单位，模拟输入为 1EU。 *)
           #tm_real := #A输入设定 * 10.0;
           #T1_SV_写 := REAL_TO_INT(#tm_real);
           #modbus_data.数据缓存区[1] := INT_TO_WORD(#T1_SV_写);
           #modbus_data.模式 := 1;
           #modbus_data.地址 := 44098;
           #modbus_data.数据长度 := 1;
       7:
           //写入地址44102
           (* 1005H-4101-44102  默认0   控制方式 0：PID；1：ON/OFF；2：手动；3：PID 过程控制 *)
           #modbus_data.数据缓存区[1] := INT_TO_WORD(#输入模式);
           #modbus_data.模式 := 1;
           #modbus_data.地址 := 44102;
           #modbus_data.数据长度 := 1;
       8:
           //写入地址44116
           (* 1013H-4115-44116  默认0   输出 2 输出量读取与写入 单位为 0.1%，写入只在手动控制模式下有效（DTC1000/2000 机种） *)
           #tm_real := #输入开度 * 10;
           #tm_int := REAL_TO_INT(#tm_real);
           #modbus_data.数据缓存区[1] := INT_TO_WORD(#tm_int);
           #modbus_data.模式 := 1;
           #modbus_data.地址 := 44116;
           #modbus_data.数据长度 := 1;
       9:
           //写入地址2068
           (* 0813H-2067-12068  读写自动调谐状态 自动调谐停止：0（预设），自动调谐开始：1 *)

           #modbus_data.数据缓存区[1] := UINT_TO_WORD(#进温AT_写字);
           #modbus_data.模式 := 1;
           #modbus_data.地址 := 2068;
           #modbus_data.数据长度 := 1;
       10:
           //写入地址2069
           (* 0814H-2068-12069  控制执行/停止设定 0：停止，1：执行（预设） *)
           #modbus_data.数据缓存区[1] := UINT_TO_WORD(#进温启停字);
           #modbus_data.模式 := 1;
           #modbus_data.地址 := 2069;
           #modbus_data.数据长度 := 1;

   END_CASE;




   #modbus_data.触发 := #当前指令ID <> #上一次指令ID;
   #上一次指令ID := #当前指令ID;



   //程序2


   #Modbus_Master_Instance(REQ := #modbus_data.触发,
                           MB_ADDR := #modbus_data.站号,
                           MODE := #modbus_data.模式,
                           DATA_ADDR := #modbus_data.地址,
                           DATA_LEN := #modbus_data.数据长度,
                           DONE => #modbus_data.完成,
                           BUSY => #modbus_data.忙碌,
                           ERROR => #modbus_data.出错,
                           STATUS => #modbus_data.故障码,
                           DATA_PTR := #modbus_data.数据缓存区);

   //程序3

   IF #modbus_data.完成 THEN
       CASE #当前指令ID OF
           1:
               //44097
               (* 1000H-4096-44097       PV 目前测量值
               （温度以 0.1 刻度为计量单位，模拟输入为 1EU。
               下列读值表示错误发生：
               8002H（32770） 输入读值尚未取得
               8003H（32771） 未接传感器
               8004H（32772） 传感器型式错误
               8006H（34774） 输入值无法测量,输入 ADC 错误
               8007H（32775） 内存无法读写） *)
               #tm_int := WORD_TO_INT(#modbus_data.数据缓存区[1]);
               #tm_real := INT_TO_REAL(#tm_int);
               #B当前量 := #tm_real / 10;
               //44098
               #tm_int := WORD_TO_INT(#modbus_data.数据缓存区[2]);
               #tm_real := INT_TO_REAL(#tm_int);
               #输入设定读 := #tm_real / 10;

           2:
               //44102
               (* 1005H-4101-44102  默认0   控制方式 0：PID；1：ON/OFF；2：手动；3：PID 过程控制 *)
               #tm_int := WORD_TO_INT(#modbus_data.数据缓存区[1]);
               #输出模式读 := #tm_int;
           3:
               (*   1009H-4105-44106  默认476 PB 比例带设定值 1 ~ 9,999, 温度单位为 0.1 度，模拟输入为 1EU
                    100AH-4106-44107  默认260 Ti 积分控制常量设定值 0 ~ 9,999
                    100BH-4107-44108  默认41 Td 微分控制常量设定值 0 ~ 9,999 *)
                    //44106
                    #tm_int := WORD_TO_INT(#modbus_data.数据缓存区[1]);
                    #进温P读 := #tm_int;
                    //44107
                    #tm_int := WORD_TO_INT(#modbus_data.数据缓存区[2]);
                    #进温I读 := #tm_int;
                    //44108
                    #tm_int := WORD_TO_INT(#modbus_data.数据缓存区[3]);
                    #进温D读 := #tm_int;
                4:
                    //44116
                    (* 1013H-4115-44116  默认0   输出 2 输出量读取与写入 单位为 0.1%，写入只在手动控制模式下有效（DTC1000/2000 机种） *)
                    #tm_int := WORD_TO_INT(#modbus_data.数据缓存区[1]);
                    #tm_real := INT_TO_REAL(#tm_int);
                    #输出开度读 := #tm_real / 10;
                5:
                    //12068
                    (* 0813H-2067-12068  读写自动调谐状态 自动调谐停止：0（预设），自动调谐开始：1 *)
                    #进温AT_读字 := WORD_TO_UINT(#modbus_data.数据缓存区[1]);
            END_CASE;
        END_IF;

        IF #modbus_data.出错 AND #当前指令ID > 0 AND #当前指令ID < 12 THEN
            #报错代码[#当前指令ID] := #modbus_data.故障码;
        END_IF;

        IF #modbus_data.完成 OR #modbus_data.出错 THEN
            #当前指令ID := #当前指令ID + 1;
        END_IF;

        IF #当前指令ID > 10 THEN
            #当前指令ID := 0;
            #上一次指令ID := 0;
            #结束 := 1;
        ELSE
            #结束 := 0;
        END_IF;

        //程序4

        IF NOT #自整定开关 THEN
            #进温AT_写字 := 0;
            #T1_P值比对1 := #进温P读;
            #T1_P值比对2 := #进温P读;
        END_IF;
        IF #自整定开关 THEN

            #进温AT_写字 := 65280;

            #T1_P值比对2 := #进温P读;
        END_IF;
        IF #T1_P值比对1 <> #T1_P值比对2 THEN
            #自整定开关 := 0;
        END_IF;

        //程序5


        IF #自整定开关 THEN
            #进温AT_写字 := 16#FF00;
        ELSE
            #进温AT_写字 := 16#0;
        END_IF;

        IF #输入开关 THEN
            #进温启停字 := 16#FF00;
        ELSE
            #进温启停字 := 16#0;
        END_IF;

       //程序6

        #输出控制P := INT_TO_REAL(#进温P读);
        #输出控制I := INT_TO_REAL(#进温I读);
        #输出控制D := INT_TO_REAL(#进温D读);

        //报警
        IF #B当前量 > #高报设置 THEN
            #高报警 := 1;
        ELSE
            #高报警 := 0;
        END_IF;

        IF #B当前量  > #高高报设置 THEN
            #高高报警 := 1;
        ELSE
            #高高报警 := 0;
        END_IF;

        IF #B当前量 < #低报设置 THEN
            #低报警 := 1;
        ELSE
            #低报警 := 0;
        END_IF;

        IF #B当前量 < #低低报设置 THEN
            #低低报警 := 1;
        ELSE
            #低低报警 := 0;
        END_IF;

        IF #B当前量 > 500 AND #B当前量 < -10 THEN
            #传感器故障 := 1;
        ELSE
            #传感器故障 := 0;
        END_IF;
END_FUNCTION_BLOCK

FUNCTION_BLOCK "Modbus_Master"   // FB641, SCL
TITLE = Modbus master communication
AUTHOR : SIMATIC
FAMILY : MODBUS
NAME : MB_MASTR
VERSION : 5.0
// stored: IsIECCheckEnabled true, SetENOAutomatically false, UDAEnableTagReadback false
   VAR_INPUT
      REQ : Bool;   // Startet die angeforderte Übertragung bei steigender Flanke / Activates the requested transmission on rising edge
      MB_ADDR : UInt;   // Modbus RTU Stationsadresse / Modbus RTU station address
      MODE : USInt;   // Bezeichnet die Art der Anforderung / Specifies the type of request
      DATA_ADDR : UDInt;   // Anfangsadresse im Slave / Starting Address in the Slave
      DATA_LEN : UInt;   // Datenlänge: Anzahl der Bits oder Wörter / Specifies the number of bits or words to be accessed
   END_VAR
   VAR_OUTPUT
      DONE : Bool;   // Anweisung beendet ohne Fehler / Instruction finished without error
      BUSY : Bool;   // Modbus Master Auftrag in Arbeit / Modbus master transaction in progress
      ERROR : Bool;   // Anweisung beendet mit Fehler / Instruction finished with error
      STATUS : Word := 16#7000;   // Detailllierte Fehlerinformation / Detailed error information
   END_VAR
   VAR_IN_OUT
      DATA_PTR : Variant;   // Referenz auf die lokale Quell- oder Zieladresse / Reference to the local source or destination address
   END_VAR
   VAR DB_SPECIFIC
      MB_State : SInt := 0;   // Internal state of the Modbus master operation
      Blocked_Proc_Timeout : Real := 3.0;   // Time to wait upon a blocked Modbus Master instance before setting inactive
      Extended_Addressing : Bool;   // Configures slave addressing; 1=double-byte adressing
      Compatibility_Mode : Bool;   // 1= data transfer for FC1, FC2 and FC15 compatible with CP341
      MB_DB { S7_SetPoint := 'True'} : P2P_MB_BASE;   // Modbus parameters
   END_VAR
   VAR
      Send_P2P { S7_SetPoint := 'True'} : Send_P2P;   // Local instance of the instruction Send_P2P
      Receive_P2P { S7_SetPoint := 'True'} : Receive_P2P;   // Local instance of the instruction Receive_P2P
      Receive_Reset { S7_SetPoint := 'True'} : Receive_Reset;   // Local instance of the instruction Receive_Reset
   END_VAR
   VAR DB_SPECIFIC
      S_PORT : Word;   // For internal use only
      S_RESP_TO : Word;   // For internal use only
      S_ICHAR_GAP : Word;   // For internal use only
      S_RETRIES : Word;   // For internal use only
      S_MB_ADDR : UInt;   // Modbus RTU station address
      S_MODE : USInt;   // Specifies the type of request
      S_DATA_ADDR : UDInt;   // Starting Address in the Slave
      S_DATA_LEN : UInt;   // Specifies the number of bits or words to be accessed
      w_retries : Word;   // For internal use only
      y_SlaveAddrHi : Byte;   // For internal use only
      y_SlaveAddrLo : Byte;   // For internal use only
      StartAddress : Word;   // For internal use only
      Value : Word;   // For internal use only
      y_FCode : Byte;   // For internal use only
   END_VAR
   VAR
      FCode_usint AT y_FCode : USInt;
   END_VAR
   VAR DB_SPECIFIC
      INTERNAL_CDATA : Array[1..257] of Byte;   // For internal use only
   END_VAR
   VAR
      FC1_2_Req AT INTERNAL_CDATA : P2P_MB_FC1_2_Req;   // For internal use only
      FC1_4_ValResp AT INTERNAL_CDATA : P2P_MB_FC1_4_ValResp;   // For internal use only
      FC3_4_Req AT INTERNAL_CDATA : P2P_MB_FC3_4_Req;   // For internal use only
      FC5_6_Req AT INTERNAL_CDATA : P2P_MB_FC5_6_Req;   // For internal use only
      FC5_6_ValResp AT INTERNAL_CDATA : P2P_MB_FC5_6_ValResp;   // For internal use only
      FC15_16_Req AT INTERNAL_CDATA : P2P_MB_FC15_16_Req;   // For internal use only
      FC11_Req AT INTERNAL_CDATA : P2P_MB_FC11_Req;   // For internal use only
      FC11_ValResp AT INTERNAL_CDATA : P2P_MB_FC11_ValResp;   // For internal use only
      FC8_Req AT INTERNAL_CDATA : P2P_MB_FC8_Req;   // For internal use only
      FCx_ErrResp AT INTERNAL_CDATA : P2P_MB_FCx_ErrResp;   // For internal use only
      MB_Header AT INTERNAL_CDATA : Struct
         free : Byte;
         SlaveAddrHi : Byte;
         SlaveAddrLo : Byte;
         FCode : Byte;
         addr : UInt;
         quantity_value : UInt;
      END_STRUCT;
      FC11 AT INTERNAL_CDATA : Struct
         free : Byte;
         SlaveAddrHi : Byte;
         SlaveAddrLo : Byte;
         FCode : Byte;
         data : Array[0..3] of Byte;
      END_STRUCT;
   END_VAR
   VAR DB_SPECIFIC
      mb_timer { S7_SetPoint := 'True'} : TON_TIME;
      TimeElapsed : Bool;
   END_VAR
BEGIN
END_FUNCTION_BLOCK

FUNCTION_BLOCK "Send_P2P"   // FB613, SCL
TITLE = Send data
AUTHOR : SIMATIC
FAMILY : Freeport
NAME : SendP2P
VERSION : 4.0
// stored: IsIECCheckEnabled true, SetENOAutomatically false, UDAEnableTagReadback false
   VAR_INPUT
      REQ : Bool;   // Startet die angeforderte Übertragung bei steigender Flanke / Activates the requested transmission on rising edge
      PORT : PORT := 16#0000;   // Kommunikationsport, Hardwarekennung / Communication port, Hardware Identifier
      BUFFER : Variant;   // Referenz auf den Sendepuffer / Reference to the send buffer
      LENGTH : UInt := 0;   // Übertragene Datenlänge in Byte / Transmitted frame length in bytes
   END_VAR
   VAR_OUTPUT
      UNIVERSAL : Bool;   // Access mode of communication module. 0 = universal, 1 = performance
      DONE : Bool;   // Anweisung beendet ohne Fehler / Instruction finished without error
      ERROR : Bool;   // Anweisung beendet mit Fehler / Instruction finished with error
      STATUS : Word := W#16#7000;   // Zusätzliche Fehlerinformation / Detailed error information
   END_VAR
   VAR
      OldPORT : PORT := 16#0000;   // Nur für internen Gebrauch / Save value for Communication port
      send_length : UInt;   // Übertragene Datenlänge in Byte / For internal use only
      max_record_len : UInt := 1026;   // Nur für internen Gebrauch / For internal use only
      max_telegram_len : UInt;
      b_e_REQ : Bool;   // Flankenbit für REQ / Edge flag for REQ
      isClassic : Bool;   // Nur für internen Gebrauch / For internal use only
      first_sent : Bool;
      y_state : SInt := 0;   // Status der Anweisung / State of instruction
      y_nr_rec : SInt;   // Nur für internen Gebrauch / Sequence number of data records
      ser_nr_old : USInt;
      ser_nr : USInt;   // Nur für internen Gebrauch / For internal use only
      module_initialized { ExternalAccessible := 'False'; ExternalVisible := 'False'; ExternalWritable := 'False'} : Bool;
   END_VAR
   VAR DB_SPECIFIC
      SendBuffer : Array[0..1026] of Byte;   // Nur für internen Gebrauch / For internal use only
   END_VAR
   VAR
      i_addr : UDInt;   // IO Adresse des Moduls / IO address of the module
      o_addr { ExternalAccessible := 'False'; ExternalVisible := 'False'; ExternalWritable := 'False'} : UDInt;
      WRREC { S7_SetPoint := 'True'} : WRREC;   // Lokale Instanz der Anweisung WRREC / Local instance of instruction WRREC
      PTP_STATUS { S7_SetPoint := 'True'} : P2P_SendGetData;   // Nur für internen Gebrauch / For internal use only
      InitTimeout { ExternalAccessible := 'False'; ExternalVisible := 'False'; ExternalWritable := 'False'; S7_SetPoint := 'True'} : TON_TIME;
   END_VAR
BEGIN
END_FUNCTION_BLOCK

FUNCTION_BLOCK "Receive_P2P"   // FB614, SCL
TITLE = Receive Data
AUTHOR : SIMATIC
FAMILY : Freeport
NAME : RcvP2P
VERSION : 4.1
// stored: IsIECCheckEnabled true, SetENOAutomatically false, UDAEnableTagReadback false
   VAR_INPUT
      PORT : PORT := 16#0000;   // Kommunikationsport, Hardwarekennung / Communication port, Hardware Identifier
      BUFFER : Variant;   // Referenz auf den Empfangspuffer / Reference to the receive buffer
   END_VAR
   VAR_OUTPUT
      UNIVERSAL : Bool;   // Access mode of communication module. 0 = universal, 1 = performance
      NDR : Bool;   // Neue Daten empfangen / New data received
      LENGTH : UInt := 16#0000;   // Länge der empfangenen Daten in Byte / Length of the current received message in bytes
      ERROR : Bool;   // Anweisung beendet mit Fehler / Instruction finished with error
      STATUS : Word := W#16#7000;   // Zusätzliche Fehlerinformation / Detailed error information
   END_VAR
   VAR
      OldPORT : PORT;   // Gespeicherter Wert für den Kommunikationsport, / Save value for Communication port
      received_length : UInt := 0;   // empfangene Länge / Received length
      y_ptp_status : SInt;   // Nur für internen Gebrauch / For internal use only
      y_state : SInt := 0;   // Status der Anweisung / State of instruction
      y_seq_nr : Byte := B#16#00;   // Sequenznummer der empfangenen Datensätze / Sequence number of data records
      safe_h1 : Byte;   // Nur für internen Gebrauch / For internal use only
      safe_h2 : Byte;   // Nur für internen Gebrauch / For internal use only
      safe_h3 : Byte;   // Nur für internen Gebrauch / For internal use only
      safe_h4 : Byte;   // Nur für internen Gebrauch / For internal use only
      isClassic : Bool;   // Nur für internen Gebrauch / For internal use only
      record_nr : Int := 49;   // Nur für internen Gebrauch / For internal use only
      offset : UDInt;   // Nur für internen Gebrauch / For internal use only
      RDREC { S7_SetPoint := 'True'} : RDREC;   // Lokale Instanz der Anweisung RDREC / Local instance of instruction RDREC
   END_VAR
   VAR DB_SPECIFIC
      ReceiveBuffer : Array[0..1027] of Byte;   // Nur für internen Gebrauch / For internal use only
   END_VAR
   VAR
      i_addr : UDInt;   // IO Adresse des Moduls / IO address of the module
      o_addr { ExternalAccessible := 'False'; ExternalVisible := 'False'; ExternalWritable := 'False'} : UDInt;
   END_VAR
BEGIN
END_FUNCTION_BLOCK

FUNCTION_BLOCK "Receive_Reset"   // FB617, SCL
TITLE = Reset Receive Buffer
AUTHOR : SIMATIC
FAMILY : Freeport
NAME : RcvRst
VERSION : 4.0
// stored: IsIECCheckEnabled false, SetENOAutomatically false, UDAEnableTagReadback false
   VAR_INPUT
      REQ : Bool;   // Löscht den Empfangspuffer mit steigender Flanke / Clears the receive buffer on rising edge
      PORT : PORT;   // Kommunikationsport, Hardwarekennung / Communication port, Hardware Identifier
   END_VAR
   VAR_OUTPUT
      DONE : Bool;   // Anweisung beendet ohne Fehler / Instruction finished without error
      ERROR : Bool;   // Anweisung beendet mit Fehler / Instruction finished with error
      STATUS : Word := W#16#7000;   // Zusätzliche Fehlerinformation / Detailed error information
   END_VAR
   VAR
      b_e_REQ : Bool;   // Flankenbit für REQ / Edge flag for REQ
      y_state : SInt;   // Status der Anweisung / State of instruction
      WRREC { S7_SetPoint := 'True'} : WRREC;   // Lokale Instanz der Anweisung WRREC / Local instance of instruction WRREC
      w_record { S7_SetPoint := 'True'} : P2P_ResetData;   // Nur für internen Gebrauch / For internal use only
   END_VAR
BEGIN
END_FUNCTION_BLOCK

FUNCTION_BLOCK "A2-数据转换ITR"   // FB56, SCL
{ S7_Optimized_Access := 'TRUE' }
VERSION : 0.1
// stored: AutoNumber true, IsIECCheckEnabled false, IsRetainMemResEnabled false, MemoryReserve 100, SetENOAutomatically false, UDAEnableTagReadback false
   VAR_INPUT
      I_ChValue : Int;   // 通道值输入
      I_Max : Int := 27648;
      I_Min : Int := 0;
      R_Max : Real;   // 仪表物理最大值(设置值)
      R_Min : Real;   // 仪表物理最小值(设置值)
      R_Edit : Real;   // 数值修订
      R_HHAlarm_Set : Real;   // 超高报警限值(设置值)
      R_HAlarm_Set : Real;   // 高报警限值(设置值)
      R_LAlarm_Set : Real;   // 低报警限值(设置值)
      R_LLAlarm_Set : Real;   // 超低报警限值(设置值)
   END_VAR
   VAR_OUTPUT
      R_Meter_Value : Real;   // 仪表实时值(输出值)
      b_HH_Alarm : Bool;   // 超高报警
      b_H_Alarm : Bool;   // 高报警
      b_L_Alarm : Bool;   // 低报警
      b_LL_Alarm : Bool;   // 超低报警
      Status : Int;   // 状态值
   END_VAR
   VAR
      input : Int;
   END_VAR
BEGIN
   (*
       数据转换AI通道值转换成仪表值
       OUT = [((FLOAT (IN) – K1)/(K2–K1)) * (HI_LIM–LO_LIM)] + LO_LIM
    *)
   (*传感器状态:0,正常;1,溢出;2:故障.*)
   IF  #I_ChValue =32767 OR #I_ChValue =-32768 THEN    //仪表故障
       #input := 0;
       #Status := 2;
   ELSIF
       #I_ChValue > 28000 AND #I_ChValue <32767 THEN   //通道溢出
       #input := 27648;
       #Status := 1;
   ELSIF #I_ChValue < -100 AND #I_ChValue >-32768 THEN   //通道溢出
       #input := 0;
       #Status := 1;
   ELSE
       #input := #I_ChValue;  //仪表正常
       #Status := 0;
   END_IF;

   #R_Meter_Value := ((INT_TO_REAL(#input)-#I_Min) / (#I_Max-#I_Min)) * (#R_Max - #R_Min) + #R_Min + #R_Edit; //仪表值计算

   IF  #R_Meter_Value >= #R_HHAlarm_Set THEN      //超高报警
       #b_HH_Alarm := 1;
   ELSE
       #b_HH_Alarm := 0;
   END_IF;

   IF #R_Meter_Value >= #R_HAlarm_Set THEN      //高报警
       #b_H_Alarm := 1;
   ELSE
       #b_H_Alarm := 0;
   END_IF;

   IF #R_Meter_Value <= #R_LLAlarm_Set THEN      //超低报警
       #b_LL_Alarm := 1;
   ELSE
       #b_LL_Alarm := 0;
   END_IF;

   IF #R_Meter_Value <= #R_LAlarm_Set THEN      //低报警
       #b_L_Alarm := 1;
   ELSE
       #b_L_Alarm := 0;
   END_IF;
END_FUNCTION_BLOCK

FUNCTION_BLOCK "A4--电机控制"   // FB6, SCL
{ S7_Optimized_Access := 'TRUE' }
VERSION : 0.1
// stored: AutoNumber true, IsIECCheckEnabled false, IsRetainMemResEnabled false, MemoryReserve 100, SetENOAutomatically false, UDAEnableTagReadback false
   VAR_INPUT
      HMI上限 : Real := 50.0;
      HMI下限 : Real;
      PLC上限 : Int := 27648;
      PLC下限 : Int := 0;
      电机报警信号 : Bool;
      电机输入模拟量 : Int;
      电机输出最小 : Real;
   END_VAR
   VAR_OUTPUT
      电机输出反馈 : Real;
      电机报警输出 : Bool;
   END_VAR
   VAR_IN_OUT
      按钮_消警按钮 : Bool;
      模式设定 : Real;
      电机控制按钮 : Bool;
      频率设定 : Real;
      电机输出Q : Bool;
      电机速度AO : Int;
      动画 : Int;
      安全停机 : Bool;
   END_VAR
   VAR
      P1 : Bool;
      TON1 : TON_TIME;
      Temp_1 { S7_SetPoint := 'True'} : Int;
      DBD1 : Real;
      DBD2 : Real;
      DBD3 : Real;
   END_VAR
BEGIN

   //手动控制--------------------------------------------------------------------------------------------------------------
   IF #模式设定 = 2.0 OR #模式设定 = 3.0  OR #模式设定 = 4.0 OR #模式设定 = 5.0  THEN
       //预热器加热手动控制
       IF #电机控制按钮 THEN
           #电机输出Q := TRUE;
           (* #电机速度AO := REAL_TO_INT(#频率设定 * 27648.0 / 50.0); *)
           #DBD1 := NORM_X_REAL(MIN := #HMI下限, VALUE := #频率设定, MAX := #HMI上限);
           #电机速度AO := SCALE_X_INT(MIN := #PLC下限, VALUE := #DBD1, MAX := #PLC上限);
       ELSE
           #电机输出Q := FALSE;
       END_IF;
   END_IF;


   // 自动启动--------------------------------------------------------------------------------------------------------------
   IF #电机输出Q THEN
       (* #电机速度AO := REAL_TO_INT(#频率设定 * 27648.0 / 50.0); *)
       #DBD2 := NORM_X_REAL(MIN := #HMI下限, VALUE := #频率设定, MAX := #HMI上限);
       #电机速度AO := SCALE_X_INT(MIN := #PLC下限, VALUE := #DBD2, MAX := #PLC上限);
   END_IF;
   IF NOT #电机输出Q THEN
       #电机速度AO := 0;
   END_IF;

   IF #电机报警输出 THEN
       #电机速度AO := 0;
       #电机控制按钮 := FALSE;
       #电机输出Q := FALSE;
   END_IF;


   IF #电机输出Q THEN
       #DBD3 := NORM_X_REAL(MIN := #PLC下限, VALUE := #电机输入模拟量, MAX := #PLC上限);
       #电机输出反馈 := SCALE_X_REAL(MIN := #HMI下限, VALUE := #DBD3, MAX := #HMI上限);
   ELSE
       #电机输出反馈 := 0;
   END_IF;
   #TON1(IN := #电机输出Q AND #电机输出反馈  < #电机输出最小,
                          PT := T#60s,
                          Q => #P1);

   IF #P1 OR #电机报警信号 THEN
       #电机报警输出 := TRUE;
   ELSE
       #电机报警输出 := FALSE;
   END_IF; 

   IF
       #模式设定 = 1 AND #电机报警输出 THEN

       #安全停机 := 1;
   END_IF;

   IF #按钮_消警按钮 THEN
       #P1 := FALSE;
       #电机报警输出 := FALSE;
   END_IF;

   IF #电机输出Q AND #频率设定 > #电机输出最小 THEN
       IF "Clock_10Hz" THEN
           #Temp_1 := #Temp_1 + 1;
       END_IF;

       IF #Temp_1 = 2 THEN
           #Temp_1 := 0;
       END_IF;
       IF #Temp_1 = 0 THEN
           #动画 := 0;
       END_IF;
       IF #Temp_1 = 1 THEN
           #动画 := 1;
       END_IF;

   END_IF;
   IF NOT #电机输出Q THEN
       #动画 := 0;
   END_IF;
END_FUNCTION_BLOCK

FUNCTION_BLOCK "A4-蠕动泵控制"   // FB9, SCL
{ S7_Optimized_Access := 'TRUE' }
VERSION : 0.1
// stored: AutoNumber true, IsIECCheckEnabled false, IsRetainMemResEnabled false, MemoryReserve 100, SetENOAutomatically false, UDAEnableTagReadback false
   VAR_INPUT
      HMI上限 : Real := 50.0;
      HMI下限 : Real;
      PLC上限 : Int := 27648;
      PLC下限 : Int := 0;
      泵报警信号 : Bool;
      泵输入电流 : Int;
   END_VAR
   VAR_OUTPUT
      泵输出反馈 : Real;
      泵报警输出 : Bool;
   END_VAR
   VAR_IN_OUT
      模式设定 : Real;
      泵控制按钮 : Bool;
      频率设定 : Real;
      泵输出Q : Bool;
      泵速度AO : Int;
      安全停机 : Bool;
      泵正反转按钮 : Bool;
      泵正反输出 : Bool;
      动画 : Int;
   END_VAR
   VAR
      Temp_1 : Int;
      DBD1 : Real;
      DBD2 : Real;
      DBD3 : Real;
   END_VAR
BEGIN

   //手动控制--------------------------------------------------------------------------------------------------------------
   IF #模式设定 = 2.0 OR #模式设定 = 3.0 OR #模式设定 = 4.0 THEN
       //预热器加热手动控制
       IF #泵控制按钮 THEN
           #泵输出Q := TRUE;
           (* #泵速度AO := REAL_TO_INT((#频率设定 - #工程下限) * (#模拟高限 - #模拟低限) / (#工程上限 - #工程下限) + #模拟低限); *)
           (* #泵速度AO := REAL_TO_INT(#频率设定 * 27648.0 / 50.0); *)
           #DBD1 := NORM_X_REAL(MIN := #HMI下限, VALUE := #频率设定, MAX := #HMI上限);
           #泵速度AO := SCALE_X_INT(MIN := #PLC下限, VALUE := #DBD1, MAX := #PLC上限);
       ELSE
           #泵输出Q := FALSE;
       END_IF;

       IF #泵正反转按钮 THEN
           #泵正反输出 := 1;
       ELSE
           #泵正反输出 := 0;
       END_IF;
   END_IF;

   //自动启动--------------------------------------------------------------------------------------------------------------


   IF #模式设定 = 1.0 THEN
       (* #泵速度AO := REAL_TO_INT((#频率设定 - #工程下限) * (#模拟高限 - #模拟低限) / (#工程上限 - #工程下限) + #模拟低限); *)
       (* #泵速度AO := REAL_TO_INT(#频率设定 * 27648.0 / 50.0); *)
       #DBD2 := NORM_X_REAL(MIN := #HMI下限, VALUE := #频率设定, MAX := #HMI上限);
       #泵速度AO := SCALE_X_INT(MIN := #PLC下限, VALUE := #DBD2, MAX := #PLC上限);



   END_IF;


   IF #泵输出Q THEN
       #DBD3 := NORM_X_REAL(MIN := #PLC下限, VALUE := #泵输入电流, MAX := #PLC上限);
       #泵输出反馈 := SCALE_X_REAL(MIN := #HMI下限, VALUE := #DBD3, MAX := #HMI上限);
   ELSE
       #泵输出反馈 := 0;
   END_IF;

   IF #泵报警信号 THEN
       #泵报警输出 := TRUE;
   ELSE
       #泵报警输出 := FALSE;
   END_IF;


   IF #泵报警信号 THEN
       #泵报警输出 := TRUE;
   ELSE
       #泵报警输出 := FALSE;
   END_IF;

   IF #泵报警输出 THEN
       #泵速度AO := 0;
       #泵控制按钮 := FALSE;
       #泵输出Q := FALSE;
   END_IF;
   IF #模式设定 = 1 AND #泵报警输出 THEN

       #安全停机 := 1;
   END_IF;


   IF #泵输出Q AND #频率设定 > 1 THEN
       IF "Clock_10Hz" THEN
           #Temp_1 := #Temp_1 + 1;
       END_IF;

       IF #Temp_1 =2 THEN
           #Temp_1 := 0;
       END_IF;
       IF #Temp_1 = 0 THEN
           #动画 := 0;
       END_IF;
       IF #Temp_1 = 1 THEN

           #动画 := 1;
       END_IF;

   END_IF;
   IF NOT #泵输出Q THEN
       #动画 := 0;
   END_IF;
END_FUNCTION_BLOCK

FUNCTION_BLOCK "A7-通信心跳块"   // FB14, SCL
{ S7_Optimized_Access := 'TRUE' }
VERSION : 0.1
// stored: AutoNumber true, IsIECCheckEnabled false, IsRetainMemResEnabled false, MemoryReserve 100, SetENOAutomatically false, UDAEnableTagReadback false
   VAR_OUTPUT
      通信失联 : Bool;
   END_VAR
   VAR_IN_OUT
      real_SC输出值 : Real;
      real_FK反馈值 : Real;
      超时时间 : Time := T#120S;
      i : Int;
   END_VAR
   VAR RETAIN
      t1 : TON_TIME;
      t2 { S7_SetPoint := 'True'} : TON_TIME;
   END_VAR
   VAR
      RT1 : R_TRIG;
   END_VAR
   VAR RETAIN
      间隔时间 : Time := T#5S;
      SC输出值 : Int;
      FK反馈值 : Int;
   END_VAR
   VAR_TEMP
      TM_FZ : Int;
   END_VAR
BEGIN
   #TM_FZ := #FK反馈值;

   #SC输出值 := REAL_TO_INT(#real_SC输出值);
   #FK反馈值 := REAL_TO_INT(#real_FK反馈值);

   #t1(IN := (#TM_FZ <> #SC输出值) ,
       PT := #超时时间,
       Q=>#通信失联);


   (* IF #t1.Q THEN
       (* #TM_FZ := 1; *)
       #SC输出值 := #SC输出值 - 1;
   END_IF; *)

   IF #TM_FZ = #SC输出值 THEN

       IF #SC输出值 MOD 2 = 0 THEN

           #SC输出值 := #SC输出值 + 1;
       ELSE

           #SC输出值 := #SC输出值 - 1;
       END_IF;

   END_IF;
END_FUNCTION_BLOCK

FUNCTION_BLOCK "A8-阀开关报警"   // FB37, SCL
{ S7_Optimized_Access := 'TRUE' }
VERSION : 0.1
// stored: AutoNumber true, IsIECCheckEnabled false, IsRetainMemResEnabled false, MemoryReserve 100, SetENOAutomatically false, UDAEnableTagReadback false
   VAR_OUTPUT
      阀开报警 : Bool;
      阀关报警 : Bool;
   END_VAR
   VAR_IN_OUT
      阀状态 : Bool;
      阀开信号 : Bool;
      阀关信号 : Bool;
   END_VAR
   VAR
      TON1 : TON_TIME;
      TON2 { S7_SetPoint := 'True'} : TON_TIME;
   END_VAR
BEGIN
   #TON1(IN := #"阀状态" AND NOT #"阀开信号",
         PT := T#10s,
         Q => #"阀开报警");
   IF NOT #"阀状态" THEN

       #"阀开报警" := FALSE;
   END_IF;


   #TON2(IN := #"阀状态" = FALSE AND NOT #"阀关信号",
         PT := T#10s,
         Q => #"阀关报警");
   IF #"阀状态" THEN

       #"阀关报警" := FALSE;
   END_IF;
END_FUNCTION_BLOCK

FUNCTION_BLOCK "B1-开式保压"   // FB34, SCL
{ S7_Optimized_Access := 'TRUE' }
VERSION : 0.1
// stored: AutoNumber true, IsIECCheckEnabled false, IsRetainMemResEnabled false, MemoryReserve 100, SetENOAutomatically false, UDAEnableTagReadback false
   VAR_OUTPUT
      MBY等待保压 : Bool;
      MBY正在充气 : Bool;
      MBY保压不佳 : Bool;
      MBY正在保压 : Bool;
      MBY保压正常 : Bool;
   END_VAR
   VAR_IN_OUT
      模式设定 : Real;
      MBY保压 : Bool;
      MQT其他阀 : Bool;
      MCQ充气阀 : Bool;
      当前阶段 : Int;
      SV保压低设定 : Real;
      SV保压高设定 : Real;
      SV保压差值 : Real;
      SV保压时 : UInt;
      SV保压分 : UInt;
      SV保压秒 : UInt;
      PV塔内压力 { ExternalAccessible := 'False'; ExternalVisible := 'False'; ExternalWritable := 'False'} : Real;
      PV保压前 { ExternalAccessible := 'False'; ExternalVisible := 'False'; ExternalWritable := 'False'} : Real;
      PV保压后 { ExternalAccessible := 'False'; ExternalVisible := 'False'; ExternalWritable := 'False'} : Real;
      PV保压当前差值 { ExternalAccessible := 'False'; ExternalVisible := 'False'; ExternalWritable := 'False'} : Real;
      PV保压时 { ExternalAccessible := 'False'; ExternalVisible := 'False'; ExternalWritable := 'False'} : UInt;
      PV保压分 { ExternalAccessible := 'False'; ExternalVisible := 'False'; ExternalWritable := 'False'} : UInt;
      PV保压秒 { ExternalAccessible := 'False'; ExternalVisible := 'False'; ExternalWritable := 'False'} : UInt;
   END_VAR
   VAR
      T_1HZ { S7_SetPoint := 'True'} : TON_TIME;
   END_VAR
BEGIN
   IF #模式设定 = 3.0 OR #模式设定 = 4.0 THEN


       IF #MBY保压 THEN

           IF #当前阶段 = 5 THEN
               #当前阶段 := 1;
           END_IF;

      ELSE
           #当前阶段 := 5; 
       END_IF;

       (* IF #MCZ重置 THEN
           #当前阶段 := 4;
           #MCZ重置 := FALSE;

       END_IF;
       *)
       CASE #当前阶段 OF
           1://开始充气
               #MQT其他阀 := 0;
               #MCQ充气阀 := 1;
               #MBY等待保压 := 0;
               #MBY正在充气 := 1;
               #MBY保压不佳 := 0;
               #MBY正在保压 := 0;
               #MBY保压正常 := 0;

               IF (#PV塔内压力 >= #SV保压低设定) AND (#PV塔内压力 <= #SV保压高设定) THEN
                   #MCQ充气阀 := 0;
                   #PV保压前 := #PV塔内压力;
                   #当前阶段 := 2;
               END_IF;
           2://时间记录
               IF #T_1HZ.Q THEN
                   #PV保压秒 += 1;
                   IF #PV保压秒 >= 60 THEN
                       #PV保压分 += 1;
                       #PV保压秒 := 0;
                       IF #PV保压分 >= 60 THEN
                           #PV保压时 += 1;
                           #PV保压分 := 0;
                       END_IF;
                   END_IF;
               END_IF;
               IF (#PV保压时 > #SV保压时) OR ((#PV保压时 = #SV保压时) AND (#PV保压分 > #SV保压分)) OR ((#PV保压时 = #SV保压时) AND (#PV保压分 = #SV保压分) AND (#PV保压秒 >= #SV保压秒)) THEN
                   #PV保压后 := #PV塔内压力;
                   #当前阶段 := 3;
               END_IF;

               #MBY等待保压 := 0;
               #MBY正在充气 := 0;
               #MBY保压不佳 := 0;
               #MBY正在保压 := 1;
               #MBY保压正常 := 0;

           3://保压结束
               #PV保压当前差值 := ABS(#PV保压前 - #PV保压后);
               #MBY保压正常 := #PV保压当前差值 < #SV保压差值;
               #MBY保压不佳 := NOT (#PV保压当前差值 < #SV保压差值);
               IF #MBY保压正常 OR #MBY保压不佳 THEN
                   #MBY正在保压 := 0;
                   #当前阶段 :=4;
               END_IF;
           4://停止保压，并记录数据



               #MBY正在充气 := 0;

               #MBY正在保压 := 0;



           5://清空数据
               #MCQ充气阀 := 0;
               #MBY保压 := 0;
               #PV保压前 := 0;
               #PV保压后 := 0;
               #PV保压时 := 0;
               #PV保压分 := 0;
               #PV保压秒 := 0;


               #MBY等待保压 := 1;
               #MBY正在充气 := 0;

               #MBY正在保压 := 0;
               #MBY保压正常 := 0;
               #MBY保压不佳 := 0;

               #PV保压当前差值 := 0.0;
       END_CASE;

       #T_1HZ(IN := NOT #T_1HZ.Q,
              PT := T#1S);
   END_IF;
END_FUNCTION_BLOCK

FUNCTION_BLOCK "B2_循环下料控制_F"   // FB38, SCL
{ S7_Optimized_Access := 'TRUE' }
VERSION : 0.1
// stored: AutoNumber true, IsIECCheckEnabled false, IsRetainMemResEnabled false, MemoryReserve 100, SetENOAutomatically false, UDAEnableTagReadback false
   VAR_INPUT
      启动按钮 : Bool;   // 启动循环下料的按钮
      停止按钮 : Bool;   // 停止循环下料的按钮
      SF上阀打开时间 : Real := 10.0;
      SF上阀关闭时间 : Real := 5.0;
      XF下阀打开时间 : Real := 10.0;
      XF下阀关闭时间 : Real := 5.0;
   END_VAR
   VAR_OUTPUT
      上阀控制 : Bool;   // 上阀控制信号 TRUE=打开
      下阀控制 : Bool;   // 下阀控制信号 TRUE=打开
      当前状态 : Int;   // 当前状态显示
      运行状态 : Bool;   // 系统运行状态
   END_VAR
   VAR
      状态 : Int := 0;   // 状态机变量：0=停止，1=上阀打开，2=上阀关闭，3=下阀打开，4=下阀关闭
      计时器 { S7_SetPoint := 'True'} : TON_TIME;   // 计时器
      上次状态 : Int := 0;   // 记录上一个状态
      启动边沿检测 { S7_SetPoint := 'True'} : R_TRIG;   // 启动按钮上升沿检测
      停止边沿检测 { S7_SetPoint := 'True'} : R_TRIG;   // 停止按钮上升沿检测
      上阀打开时间 : Time;   // 上阀打开持续时间 默认10秒
      上阀关闭时间 : Time;   // 上阀关闭持续时间 默认5秒
      下阀打开时间 : Time;   // 下阀打开持续时间 默认10秒
      下阀关闭时间 : Time;   // 下阀关闭持续时间 默认5秒
   END_VAR
BEGIN
       // 检测启动按钮上升沿
       // REAL_MS_TO_TIME := DINT_TO_TIME(REAL_TO_DINT(IN_REAL * 1000.0));
       // REAL_MS_TO_TIME := DINT_TO_TIME(REAL_TO_DINT(IN_REAL));
       #上阀打开时间 := DINT_TO_TIME(REAL_TO_DINT(#SF上阀打开时间 * 1000.0));
       #上阀关闭时间 := DINT_TO_TIME(REAL_TO_DINT(#SF上阀关闭时间 * 1000.0));
       #下阀打开时间 := DINT_TO_TIME(REAL_TO_DINT(#XF下阀打开时间 * 1000.0));
       #下阀关闭时间 := DINT_TO_TIME(REAL_TO_DINT(#XF下阀关闭时间 * 1000.0));

      // TotalMS := TIME_TO_DINT(IN_TIME); // 转换为毫秒
       // TIME_TO_REAL_MS := DINT_TO_REAL(TIME_TO_DINT(IN_TIME));
       // TIME_TO_REAL_S := DINT_TO_REAL(TIME_TO_DINT(IN_TIME)) / 1000.0;
       #启动边沿检测(CLK := #启动按钮);

       // 检测停止按钮上升沿
       #停止边沿检测(CLK := #停止按钮);

       // 处理启动/停止
       IF #停止边沿检测.Q THEN
           #状态 := 0;  // 停止
           #运行状态 := FALSE;
       ELSIF #启动边沿检测.Q AND #状态 = 0 THEN
           #状态 := 1;  // 启动，从上阀打开开始
           #运行状态 := TRUE;
       END_IF;

       // 状态机逻辑
       CASE #状态 OF
           0:  // 停止状态
               #上阀控制 := FALSE;
               #下阀控制 := FALSE;
               #计时器(IN := FALSE,
                    PT := T#0S);

           1:  // 状态1：上阀打开
               #上阀控制 := TRUE;
               #下阀控制 := FALSE;

               // 如果状态刚刚变化，重置计时器
               IF #上次状态 <> #状态 THEN
                   #计时器(IN := FALSE,
                        PT := #上阀打开时间);
                   #上次状态 := #状态;
               END_IF;

               // 启动计时器
               #计时器(IN := TRUE,
                    PT := #上阀打开时间);

               // 当计时器到达设定时间，切换到下一个状态
               IF #计时器.Q THEN
                   #状态 := 2;  // 切换到上阀关闭状态
               END_IF;

           2:  // 状态2：上阀关闭
               #上阀控制 := FALSE;
               #下阀控制 := FALSE;

               // 如果状态刚刚变化，重置计时器
               IF #上次状态 <> #状态 THEN
                   #计时器(IN := FALSE,
                        PT := #上阀关闭时间);
                   #上次状态 := #状态;
               END_IF;

               // 启动计时器
               #计时器(IN := TRUE,
                    PT := #上阀关闭时间);

               // 当计时器到达设定时间，切换到下一个状态
               IF #计时器.Q THEN
                   #状态 := 3;  // 切换到下阀打开状态
               END_IF;

           3:  // 状态3：下阀打开
               #上阀控制 := FALSE;
               #下阀控制 := TRUE;

               // 如果状态刚刚变化，重置计时器
               IF #上次状态 <> #状态 THEN
                   #计时器(IN := FALSE,
                        PT := #下阀打开时间);
                   #上次状态 := #状态;
               END_IF;

               // 启动计时器
               #计时器(IN := TRUE,
                    PT := #下阀打开时间);

               // 当计时器到达设定时间，切换到下一个状态
               IF #计时器.Q THEN
                   #状态 := 4;  // 切换到下阀关闭状态
               END_IF;

           4:  // 状态4：下阀关闭
               #上阀控制 := FALSE;
               #下阀控制 := FALSE;

               // 如果状态刚刚变化，重置计时器
               IF #上次状态 <> #状态 THEN
                   #计时器(IN := FALSE,
                        PT := #下阀关闭时间);
                   #上次状态 := #状态;
               END_IF;

               // 启动计时器
               #计时器(IN := TRUE,
                    PT := #下阀关闭时间);

               // 当计时器到达设定时间，切换回第一个状态
               IF #计时器.Q THEN
                   #状态 := 1;  // 返回上阀打开状态，完成一个循环
               END_IF;

